LIN {X 0.115,Y -679.979,Z 928.446,A 0.000,B 0.000,C 90.000,E1 296.309} C_DIS
LIN {X -0.394,Y -681.905,Z 928.440,A 0.000,B 0.000,C 90.000,E1 295.155} C_DIS
LIN {X 0.151,Y -683.265,Z 928.434,A 0.000,B 0.000,C 90.000,E1 294.155} C_DIS
LIN {X 0.090,Y -684.389,Z 928.429,A 0.000,B 0.000,C 90.000,E1 293.206} C_DIS
LIN {X -0.388,Y -684.559,Z 928.426,A 0.000,B 0.000,C 90.000,E1 292.770} C_DIS
LIN {X -0.179,Y -684.600,Z 928.425,A 0.000,B 0.000,C 90.000,E1 292.514} C_DIS
LIN {X -0.022,Y -683.786,Z 928.422,A 0.000,B 0.000,C 90.000,E1 292.025} C_DIS
LIN {X 0.182,Y -683.293,Z 928.421,A 0.000,B 0.000,C 90.000,E1 291.770} C_DIS
LIN {X 0.031,Y -682.793,Z 928.420,A 0.000,B 0.000,C 90.000,E1 291.663} C_DIS
LIN {X 0.133,Y -682.008,Z 928.420,A 0.000,B 0.000,C 90.000,E1 291.535} C_DIS
LIN {X -0.294,Y -677.350,Z 928.417,A 0.000,B 0.000,C 90.000,E1 291.099} C_DIS
LIN {X -0.020,Y -676.163,Z 928.417,A 0.000,B 0.000,C 90.000,E1 290.972} C_DIS
LIN {X -0.216,Y -672.859,Z 928.415,A 0.000,B 0.000,C 90.000,E1 290.791} C_DIS
LIN {X 0.088,Y -663.665,Z 928.413,A 0.000,B 0.000,C 90.000,E1 290.248} C_DIS
LIN {X -0.132,Y -662.068,Z 928.412,A 0.000,B 0.000,C 90.000,E1 290.120} C_DIS
LIN {X -0.175,Y -662.057,Z 928.412,A 0.000,B 0.000,C 90.000,E1 290.120} C_DIS
LIN {X -0.103,Y -661.805,Z 928.411,A 0.000,B 0.000,C 90.000,E1 289.939} C_DIS
LIN {X 0.025,Y -662.671,Z 928.408,A 0.000,B 0.000,C 90.000,E1 289.504} C_DIS
LIN {X -0.122,Y -665.204,Z 928.405,A 0.000,B 0.000,C 90.000,E1 288.906} C_DIS
LIN {X -0.022,Y -671.493,Z 928.398,A 0.000,B 0.000,C 90.000,E1 287.692} C_DIS
LIN {X -0.225,Y -674.954,Z 928.394,A 0.000,B 0.000,C 90.000,E1 286.985} C_DIS
LIN {X -0.146,Y -676.936,Z 928.392,A 0.000,B 0.000,C 90.000,E1 286.496} C_DIS
LIN {X -0.291,Y -679.446,Z 928.388,A 0.000,B 0.000,C 90.000,E1 285.788} C_DIS
LIN {X -0.230,Y -681.318,Z 928.384,A 0.000,B 0.000,C 90.000,E1 285.064} C_DIS
LIN {X 0.301,Y -683.455,Z 928.378,A 0.000,B 0.000,C 90.000,E1 284.064} C_DIS
LIN {X 0.201,Y -685.101,Z 928.373,A 0.000,B 0.000,C 90.000,E1 283.119} C_DIS
LIN {X 0.136,Y -686.117,Z 928.369,A 0.000,B 0.000,C 90.000,E1 282.411} C_DIS
LIN {X -0.066,Y -686.891,Z 928.365,A 0.000,B 0.000,C 90.000,E1 281.715} C_DIS
LIN {X -0.102,Y -687.225,Z 928.362,A 0.000,B 0.000,C 90.000,E1 281.243} C_DIS
LIN {X -0.268,Y -687.192,Z 928.360,A 0.000,B 0.000,C 90.000,E1 280.782} C_DIS
LIN {X 0.349,Y -686.686,Z 928.356,A 0.000,B 0.000,C 90.000,E1 280.018} C_DIS
LIN {X 0.186,Y -685.782,Z 928.353,A 0.000,B 0.000,C 90.000,E1 279.557} C_DIS
LIN {X 0.022,Y -684.420,Z 928.351,A 0.000,B 0.000,C 90.000,E1 279.095} C_DIS
LIN {X -0.009,Y -683.605,Z 928.349,A 0.000,B 0.000,C 90.000,E1 278.859} C_DIS
LIN {X -0.183,Y -681.661,Z 928.347,A 0.000,B 0.000,C 90.000,E1 278.398} C_DIS
LIN {X 0.124,Y -676.310,Z 928.341,A 0.000,B 0.000,C 90.000,E1 277.296} C_DIS
LIN {X -0.253,Y -671.792,Z 928.336,A 0.000,B 0.000,C 90.000,E1 276.486} C_DIS
LIN {X 0.079,Y -668.243,Z 928.333,A 0.000,B 0.000,C 90.000,E1 275.853} C_DIS
LIN {X -0.280,Y -664.000,Z 928.329,A 0.000,B 0.000,C 90.000,E1 275.277} C_DIS
LIN {X 0.079,Y -660.284,Z 928.327,A 0.000,B 0.000,C 90.000,E1 274.759} C_DIS
LIN {X 0.260,Y -655.075,Z 928.323,A 0.000,B 0.000,C 90.000,E1 274.131} C_DIS
LIN {X -0.097,Y -650.616,Z 928.320,A 0.000,B 0.000,C 90.000,E1 273.669} C_DIS
LIN {X 0.179,Y -644.503,Z 928.317,A 0.000,B 0.000,C 90.000,E1 273.037} C_DIS
LIN {X 0.014,Y -637.880,Z 928.314,A 0.000,B 0.000,C 90.000,E1 272.465} C_DIS
LIN {X 0.210,Y -630.842,Z 928.311,A 0.000,B 0.000,C 90.000,E1 271.892} C_DIS
LIN {X 0.177,Y -623.249,Z 928.308,A 0.000,B 0.000,C 90.000,E1 271.375} C_DIS
LIN {X -0.081,Y -615.438,Z 928.305,A 0.000,B 0.000,C 90.000,E1 270.917} C_DIS
LIN {X 0.026,Y -610.795,Z 928.304,A 0.000,B 0.000,C 90.000,E1 270.630} C_DIS
LIN {X 0.019,Y -604.204,Z 928.302,A 0.000,B 0.000,C 90.000,E1 270.286} C_DIS
LIN {X 0.254,Y -597.487,Z 928.300,A 0.000,B 0.000,C 90.000,E1 269.943} C_DIS
LIN {X 0.204,Y -590.404,Z 928.298,A 0.000,B 0.000,C 90.000,E1 269.656} C_DIS
LIN {X -0.043,Y -585.027,Z 928.297,A 0.000,B 0.000,C 90.000,E1 269.484} C_DIS
LIN {X -0.044,Y -577.197,Z 928.296,A 0.000,B 0.000,C 90.000,E1 269.255} C_DIS
LIN {X 0.274,Y -571.267,Z 928.295,A 0.000,B 0.000,C 90.000,E1 269.083} C_DIS
LIN {X -0.226,Y -565.261,Z 928.294,A 0.000,B 0.000,C 90.000,E1 269.026} C_DIS
LIN {X 0.072,Y -557.427,Z 928.294,A 0.000,B 0.000,C 90.000,E1 268.912} C_DIS
LIN {X 0.257,Y -552.326,Z 928.294,A 0.000,B 0.000,C 90.000,E1 268.854} C_DIS
LIN {X -0.168,Y -550.890,Z 928.294,A 0.000,B 0.000,C 90.000,E1 268.854} C_DIS
LIN {X -0.201,Y -550.829,Z 928.294,A 0.000,B 0.000,C 90.000,E1 268.854} C_DIS
LIN {X 0.151,Y -550.326,Z 928.293,A 0.000,B 0.000,C 90.000,E1 268.740} C_DIS
LIN {X 0.155,Y -546.076,Z 928.290,A 0.000,B 0.000,C 90.000,E1 268.224} C_DIS
LIN {X 0.133,Y -544.236,Z 928.289,A 0.000,B 0.000,C 90.000,E1 268.051} C_DIS
LIN {X 0.091,Y -544.197,Z 928.289,A 0.000,B 0.000,C 90.000,E1 268.051} C_DIS
LIN {X -0.037,Y -543.551,Z 928.288,A 0.000,B 0.000,C 90.000,E1 267.822} C_DIS
LIN {X 0.095,Y -542.151,Z 928.281,A 0.000,B 0.000,C 90.000,E1 266.617} C_DIS
LIN {X -0.169,Y -540.126,Z 928.267,A 0.000,B 0.000,C 90.000,E1 264.090} C_DIS
LIN {X 0.086,Y -538.982,Z 928.258,A 0.000,B 0.000,C 90.000,E1 262.356} C_DIS
LIN {X -0.281,Y -537.936,Z 928.250,A 0.000,B 0.000,C 90.000,E1 260.971} C_DIS
LIN {X -0.091,Y -537.174,Z 928.245,A 0.000,B 0.000,C 90.000,E1 260.095} C_DIS
LIN {X 0.097,Y -536.165,Z 928.240,A 0.000,B 0.000,C 90.000,E1 259.218} C_DIS
LIN {X 0.064,Y -532.655,Z 928.226,A 0.000,B 0.000,C 90.000,E1 256.645} C_DIS
LIN {X 0.087,Y -530.180,Z 928.215,A 0.000,B 0.000,C 90.000,E1 254.629} C_DIS
LIN {X 0.023,Y -528.110,Z 928.205,A 0.000,B 0.000,C 90.000,E1 252.906} C_DIS
LIN {X 0.055,Y -526.299,Z 928.197,A 0.000,B 0.000,C 90.000,E1 251.456} C_DIS
LIN {X 0.053,Y -523.295,Z 928.184,A 0.000,B 0.000,C 90.000,E1 249.135} C_DIS
LIN {X -0.153,Y -520.997,Z 928.174,A 0.000,B 0.000,C 90.000,E1 247.411} C_DIS
LIN {X 0.115,Y -518.888,Z 928.166,A 0.000,B 0.000,C 90.000,E1 245.921} C_DIS
LIN {X 0.212,Y -516.133,Z 928.157,A 0.000,B 0.000,C 90.000,E1 244.152} C_DIS
LIN {X 0.121,Y -513.836,Z 928.148,A 0.000,B 0.000,C 90.000,E1 242.692} C_DIS
LIN {X -0.235,Y -511.323,Z 928.140,A 0.000,B 0.000,C 90.000,E1 241.257} C_DIS
LIN {X -0.017,Y -509.278,Z 928.134,A 0.000,B 0.000,C 90.000,E1 240.049} C_DIS
LIN {X 0.242,Y -506.592,Z 928.125,A 0.000,B 0.000,C 90.000,E1 238.535} C_DIS
LIN {X -0.036,Y -504.197,Z 928.119,A 0.000,B 0.000,C 90.000,E1 237.375} C_DIS
LIN {X 0.071,Y -501.549,Z 928.112,A 0.000,B 0.000,C 90.000,E1 236.167} C_DIS
LIN {X -0.116,Y -496.120,Z 928.099,A 0.000,B 0.000,C 90.000,E1 233.783} C_DIS
LIN {X -0.109,Y -491.517,Z 928.087,A 0.000,B 0.000,C 90.000,E1 231.662} C_DIS
LIN {X 0.122,Y -489.459,Z 928.082,A 0.000,B 0.000,C 90.000,E1 230.723} C_DIS
LIN {X -0.248,Y -485.323,Z 928.072,A 0.000,B 0.000,C 90.000,E1 228.933} C_DIS
LIN {X -0.204,Y -481.829,Z 928.063,A 0.000,B 0.000,C 90.000,E1 227.391} C_DIS
LIN {X 0.219,Y -477.697,Z 928.053,A 0.000,B 0.000,C 90.000,E1 225.486} C_DIS
LIN {X -0.003,Y -475.046,Z 928.046,A 0.000,B 0.000,C 90.000,E1 224.271} C_DIS
LIN {X -0.061,Y -470.852,Z 928.036,A 0.000,B 0.000,C 90.000,E1 222.405} C_DIS
LIN {X -0.047,Y -468.121,Z 928.029,A 0.000,B 0.000,C 90.000,E1 221.148} C_DIS
LIN {X -0.019,Y -461.957,Z 928.013,A 0.000,B 0.000,C 90.000,E1 218.302} C_DIS
LIN {X -0.020,Y -459.252,Z 928.006,A 0.000,B 0.000,C 90.000,E1 217.030} C_DIS
LIN {X -0.056,Y -455.812,Z 927.997,A 0.000,B 0.000,C 90.000,E1 215.438} C_DIS
LIN {X 0.030,Y -451.538,Z 927.986,A 0.000,B 0.000,C 90.000,E1 213.499} C_DIS
LIN {X 0.151,Y -447.320,Z 927.975,A 0.000,B 0.000,C 90.000,E1 211.544} C_DIS
LIN {X 0.105,Y -440.899,Z 927.959,A 0.000,B 0.000,C 90.000,E1 208.615} C_DIS
LIN {X -0.144,Y -438.025,Z 927.952,A 0.000,B 0.000,C 90.000,E1 207.334} C_DIS
LIN {X -0.020,Y -434.378,Z 927.943,A 0.000,B 0.000,C 90.000,E1 205.668} C_DIS
LIN {X 0.038,Y -429.286,Z 927.930,A 0.000,B 0.000,C 90.000,E1 203.334} C_DIS
LIN {X -0.174,Y -426.387,Z 927.922,A 0.000,B 0.000,C 90.000,E1 202.025} C_DIS
LIN {X 0.144,Y -422.679,Z 927.913,A 0.000,B 0.000,C 90.000,E1 200.301} C_DIS
LIN {X -0.033,Y -416.572,Z 927.896,A 0.000,B 0.000,C 90.000,E1 197.275} C_DIS
LIN {X -0.090,Y -414.522,Z 927.890,A 0.000,B 0.000,C 90.000,E1 196.260} C_DIS
LIN {X -0.012,Y -410.975,Z 927.881,A 0.000,B 0.000,C 90.000,E1 194.537} C_DIS
LIN {X -0.124,Y -408.214,Z 927.873,A 0.000,B 0.000,C 90.000,E1 193.175} C_DIS
LIN {X 0.121,Y -403.378,Z 927.860,A 0.000,B 0.000,C 90.000,E1 190.715} C_DIS
LIN {X 0.076,Y -398.649,Z 927.846,A 0.000,B 0.000,C 90.000,E1 188.276} C_DIS
LIN {X 0.182,Y -393.790,Z 927.832,A 0.000,B 0.000,C 90.000,E1 185.796} C_DIS
LIN {X 0.017,Y -388.588,Z 927.817,A 0.000,B 0.000,C 90.000,E1 182.980} C_DIS
LIN {X 0.071,Y -382.269,Z 927.795,A 0.000,B 0.000,C 90.000,E1 179.026} C_DIS
LIN {X 0.116,Y -381.021,Z 927.789,A 0.000,B 0.000,C 90.000,E1 177.936} C_DIS
LIN {X 0.130,Y -380.155,Z 927.783,A 0.000,B 0.000,C 90.000,E1 176.849} C_DIS
LIN {X -0.103,Y -380.088,Z 927.779,A 0.000,B 0.000,C 90.000,E1 176.159} C_DIS
LIN {X 0.044,Y -380.506,Z 927.775,A 0.000,B 0.000,C 90.000,E1 175.412} C_DIS
LIN {X -0.055,Y -381.032,Z 927.773,A 0.000,B 0.000,C 90.000,E1 175.065} C_DIS
LIN {X -0.179,Y -382.141,Z 927.770,A 0.000,B 0.000,C 90.000,E1 174.609} C_DIS
LIN {X -0.206,Y -384.369,Z 927.767,A 0.000,B 0.000,C 90.000,E1 174.033} C_DIS
LIN {X -0.085,Y -386.614,Z 927.765,A 0.000,B 0.000,C 90.000,E1 173.628} C_DIS
LIN {X -0.161,Y -389.018,Z 927.763,A 0.000,B 0.000,C 90.000,E1 173.280} C_DIS
LIN {X -0.073,Y -391.403,Z 927.761,A 0.000,B 0.000,C 90.000,E1 172.989} C_DIS
LIN {X 0.127,Y -395.578,Z 927.759,A 0.000,B 0.000,C 90.000,E1 172.534} C_DIS
LIN {X 0.119,Y -403.599,Z 927.755,A 0.000,B 0.000,C 90.000,E1 171.894} C_DIS
LIN {X 0.216,Y -413.105,Z 927.751,A 0.000,B 0.000,C 90.000,E1 171.197} C_DIS
LIN {X -0.058,Y -424.372,Z 927.747,A 0.000,B 0.000,C 90.000,E1 170.387} C_DIS
LIN {X 0.074,Y -433.736,Z 927.742,A 0.000,B 0.000,C 90.000,E1 169.634} C_DIS
LIN {X -0.122,Y -438.390,Z 927.740,A 0.000,B 0.000,C 90.000,E1 169.285} C_DIS
LIN {X -0.153,Y -445.924,Z 927.737,A 0.000,B 0.000,C 90.000,E1 168.634} C_DIS
LIN {X 0.139,Y -453.234,Z 927.733,A 0.000,B 0.000,C 90.000,E1 167.937} C_DIS
LIN {X -0.032,Y -461.903,Z 927.728,A 0.000,B 0.000,C 90.000,E1 167.117} C_DIS
LIN {X -0.138,Y -468.940,Z 927.724,A 0.000,B 0.000,C 90.000,E1 166.408} C_DIS
LIN {X -0.197,Y -476.850,Z 927.719,A 0.000,B 0.000,C 90.000,E1 165.519} C_DIS
LIN {X -0.177,Y -486.002,Z 927.714,A 0.000,B 0.000,C 90.000,E1 164.448} C_DIS
LIN {X -0.166,Y -491.991,Z 927.709,A 0.000,B 0.000,C 90.000,E1 163.685} C_DIS
LIN {X 0.049,Y -499.996,Z 927.703,A 0.000,B 0.000,C 90.000,E1 162.598} C_DIS
LIN {X 0.223,Y -512.447,Z 927.693,A 0.000,B 0.000,C 90.000,E1 160.786} C_DIS
LIN {X 0.067,Y -520.436,Z 927.687,A 0.000,B 0.000,C 90.000,E1 159.625} C_DIS
LIN {X 0.022,Y -527.959,Z 927.680,A 0.000,B 0.000,C 90.000,E1 158.465} C_DIS
LIN {X 0.077,Y -535.176,Z 927.674,A 0.000,B 0.000,C 90.000,E1 157.305} C_DIS
LIN {X 0.045,Y -544.769,Z 927.665,A 0.000,B 0.000,C 90.000,E1 155.741} C_DIS
LIN {X -0.333,Y -550.536,Z 927.660,A 0.000,B 0.000,C 90.000,E1 154.793} C_DIS
LIN {X -0.120,Y -557.640,Z 927.653,A 0.000,B 0.000,C 90.000,E1 153.512} C_DIS
LIN {X 0.211,Y -564.128,Z 927.646,A 0.000,B 0.000,C 90.000,E1 152.231} C_DIS
LIN {X -0.076,Y -566.272,Z 927.644,A 0.000,B 0.000,C 90.000,E1 151.847} C_DIS
LIN {X -0.092,Y -574.176,Z 927.634,A 0.000,B 0.000,C 90.000,E1 150.205} C_DIS
LIN {X -0.226,Y -579.539,Z 927.628,A 0.000,B 0.000,C 90.000,E1 148.997} C_DIS
LIN {X -0.226,Y -581.876,Z 927.625,A 0.000,B 0.000,C 90.000,E1 148.456} C_DIS
LIN {X -0.128,Y -588.414,Z 927.616,A 0.000,B 0.000,C 90.000,E1 146.834} C_DIS
LIN {X 0.007,Y -592.718,Z 927.610,A 0.000,B 0.000,C 90.000,E1 145.754} C_DIS
LIN {X 0.045,Y -596.901,Z 927.604,A 0.000,B 0.000,C 90.000,E1 144.689} C_DIS
LIN {X -0.094,Y -599.878,Z 927.599,A 0.000,B 0.000,C 90.000,E1 143.909} C_DIS
LIN {X 0.084,Y -605.610,Z 927.591,A 0.000,B 0.000,C 90.000,E1 142.316} C_DIS
LIN {X -0.193,Y -612.532,Z 927.581,A 0.000,B 0.000,C 90.000,E1 140.517} C_DIS
LIN {X 0.155,Y -618.534,Z 927.572,A 0.000,B 0.000,C 90.000,E1 138.933} C_DIS
LIN {X 0.089,Y -628.640,Z 927.558,A 0.000,B 0.000,C 90.000,E1 136.377} C_DIS
LIN {X 0.058,Y -632.754,Z 927.552,A 0.000,B 0.000,C 90.000,E1 135.364} C_DIS
LIN {X -0.115,Y -638.687,Z 927.544,A 0.000,B 0.000,C 90.000,E1 133.866} C_DIS
LIN {X -0.004,Y -642.636,Z 927.538,A 0.000,B 0.000,C 90.000,E1 132.852} C_DIS
LIN {X -0.049,Y -650.428,Z 927.527,A 0.000,B 0.000,C 90.000,E1 130.862} C_DIS
LIN {X -0.261,Y -655.186,Z 927.520,A 0.000,B 0.000,C 90.000,E1 129.644} C_DIS
LIN {X 0.130,Y -661.759,Z 927.511,A 0.000,B 0.000,C 90.000,E1 127.890} C_DIS
LIN {X 0.166,Y -667.284,Z 927.503,A 0.000,B 0.000,C 90.000,E1 126.423} C_DIS
LIN {X -0.080,Y -671.674,Z 927.496,A 0.000,B 0.000,C 90.000,E1 125.231} C_DIS
LIN {X 0.148,Y -674.922,Z 927.490,A 0.000,B 0.000,C 90.000,E1 124.246} C_DIS
LIN {X 0.438,Y -677.247,Z 927.486,A 0.000,B 0.000,C 90.000,E1 123.499} C_DIS
LIN {X -0.183,Y -679.386,Z 927.482,A 0.000,B 0.000,C 90.000,E1 122.832} C_DIS
LIN {X 0.323,Y -682.523,Z 927.476,A 0.000,B 0.000,C 90.000,E1 121.592} C_DIS
LIN {X -0.043,Y -684.633,Z 927.470,A 0.000,B 0.000,C 90.000,E1 120.669} C_DIS
LIN {X -0.001,Y -686.108,Z 927.466,A 0.000,B 0.000,C 90.000,E1 119.951} C_DIS
LIN {X 0.019,Y -687.763,Z 927.461,A 0.000,B 0.000,C 90.000,E1 118.999} C_DIS
LIN {X 0.089,Y -688.867,Z 927.457,A 0.000,B 0.000,C 90.000,E1 118.281} C_DIS
LIN {X 0.084,Y -689.911,Z 927.452,A 0.000,B 0.000,C 90.000,E1 117.334} C_DIS
LIN {X -0.203,Y -690.487,Z 927.447,A 0.000,B 0.000,C 90.000,E1 116.411} C_DIS
LIN {X 0.206,Y -690.666,Z 927.443,A 0.000,B 0.000,C 90.000,E1 115.668} C_DIS
LIN {X 0.241,Y -690.715,Z 927.438,A 0.000,B 0.000,C 90.000,E1 114.719} C_DIS
LIN {X 0.038,Y -690.480,Z 927.434,A 0.000,B 0.000,C 90.000,E1 114.027} C_DIS
LIN {X -0.125,Y -690.060,Z 927.431,A 0.000,B 0.000,C 90.000,E1 113.567} C_DIS
LIN {X -0.168,Y -689.627,Z 927.430,A 0.000,B 0.000,C 90.000,E1 113.334} C_DIS
LIN {X 0.290,Y -688.240,Z 927.427,A 0.000,B 0.000,C 90.000,E1 112.823} C_DIS
LIN {X 0.137,Y -687.716,Z 927.426,A 0.000,B 0.000,C 90.000,E1 112.717} C_DIS
LIN {X -0.059,Y -684.321,Z 927.424,A 0.000,B 0.000,C 90.000,E1 112.259} C_DIS
LIN {X -0.211,Y -683.240,Z 927.423,A 0.000,B 0.000,C 90.000,E1 112.153} C_DIS
LIN {X -0.108,Y -681.860,Z 927.422,A 0.000,B 0.000,C 90.000,E1 112.025} C_DIS
LIN {X -0.005,Y -679.584,Z 927.422,A 0.000,B 0.000,C 90.000,E1 111.897} C_DIS
LIN {X 0.194,Y -674.984,Z 927.421,A 0.000,B 0.000,C 90.000,E1 111.716} C_DIS
LIN {X 0.300,Y -669.777,Z 927.420,A 0.000,B 0.000,C 90.000,E1 111.535} C_DIS
LIN {X -0.371,Y -666.947,Z 927.419,A 0.000,B 0.000,C 90.000,E1 111.535} C_DIS
LIN {X -0.229,Y -659.882,Z 927.419,A 0.000,B 0.000,C 90.000,E1 111.461} C_DIS
LIN {X 0.340,Y -652.708,Z 927.419,A 0.000,B 0.000,C 90.000,E1 111.408} C_DIS
LIN {X 0.295,Y -643.253,Z 927.419,A 0.000,B 0.000,C 90.000,E1 111.408} C_DIS
LIN {X -0.011,Y -638.058,Z 927.419,A 0.000,B 0.000,C 90.000,E1 111.408} C_DIS
LIN {X 0.198,Y -634.455,Z 927.419,A 0.000,B 0.000,C 90.000,E1 111.354} C_DIS
LIN {X 0.110,Y -629.194,Z 927.418,A 0.000,B 0.000,C 90.000,E1 111.280} C_DIS
LIN {X -0.190,Y -621.802,Z 927.417,A 0.000,B 0.000,C 90.000,E1 111.153} C_DIS
LIN {X 0.094,Y -614.447,Z 927.416,A 0.000,B 0.000,C 90.000,E1 110.918} C_DIS
LIN {X -0.134,Y -606.224,Z 927.414,A 0.000,B 0.000,C 90.000,E1 110.610} C_DIS
LIN {X -0.176,Y -603.378,Z 927.414,A 0.000,B 0.000,C 90.000,E1 110.482} C_DIS
LIN {X 0.115,Y -598.239,Z 927.412,A 0.000,B 0.000,C 90.000,E1 110.174} C_DIS
LIN {X -0.185,Y -590.045,Z 927.409,A 0.000,B 0.000,C 90.000,E1 109.685} C_DIS
LIN {X -0.322,Y -583.118,Z 927.407,A 0.000,B 0.000,C 90.000,E1 109.214} C_DIS
LIN {X -0.218,Y -578.724,Z 927.405,A 0.000,B 0.000,C 90.000,E1 108.906} C_DIS
LIN {X 0.107,Y -571.680,Z 927.403,A 0.000,B 0.000,C 90.000,E1 108.489} C_DIS
LIN {X 0.028,Y -564.876,Z 927.401,A 0.000,B 0.000,C 90.000,E1 108.181} C_DIS
LIN {X 0.222,Y -557.773,Z 927.399,A 0.000,B 0.000,C 90.000,E1 107.873} C_DIS
LIN {X -0.079,Y -554.844,Z 927.399,A 0.000,B 0.000,C 90.000,E1 107.764} C_DIS
LIN {X 0.048,Y -552.961,Z 927.398,A 0.000,B 0.000,C 90.000,E1 107.583} C_DIS
LIN {X 0.010,Y -552.942,Z 927.398,A 0.000,B 0.000,C 90.000,E1 107.583} C_DIS
LIN {X 0.136,Y -552.516,Z 927.396,A 0.000,B 0.000,C 90.000,E1 107.330} C_DIS
LIN {X 0.117,Y -552.658,Z 927.392,A 0.000,B 0.000,C 90.000,E1 106.622} C_DIS
LIN {X -0.196,Y -553.186,Z 927.386,A 0.000,B 0.000,C 90.000,E1 105.536} C_DIS
LIN {X 0.116,Y -553.904,Z 927.377,A 0.000,B 0.000,C 90.000,E1 103.828} C_DIS
LIN {X 0.034,Y -555.068,Z 927.366,A 0.000,B 0.000,C 90.000,E1 101.883} C_DIS
LIN {X -0.115,Y -556.765,Z 927.354,A 0.000,B 0.000,C 90.000,E1 99.670} C_DIS
LIN {X -0.083,Y -557.816,Z 927.346,A 0.000,B 0.000,C 90.000,E1 98.276} C_DIS
LIN {X -0.112,Y -558.880,Z 927.338,A 0.000,B 0.000,C 90.000,E1 96.891} C_DIS
LIN {X -0.048,Y -559.931,Z 927.329,A 0.000,B 0.000,C 90.000,E1 95.220} C_DIS
LIN {X -0.098,Y -560.701,Z 927.321,A 0.000,B 0.000,C 90.000,E1 93.841} C_DIS
LIN {X -0.168,Y -561.417,Z 927.314,A 0.000,B 0.000,C 90.000,E1 92.465} C_DIS
LIN {X -0.127,Y -562.099,Z 927.304,A 0.000,B 0.000,C 90.000,E1 90.802} C_DIS
LIN {X 0.278,Y -562.437,Z 927.298,A 0.000,B 0.000,C 90.000,E1 89.656} C_DIS
LIN {X 0.222,Y -562.782,Z 927.291,A 0.000,B 0.000,C 90.000,E1 88.282} C_DIS
LIN {X 0.184,Y -563.045,Z 927.283,A 0.000,B 0.000,C 90.000,E1 86.906} C_DIS
LIN {X 0.088,Y -563.269,Z 927.277,A 0.000,B 0.000,C 90.000,E1 85.812} C_DIS
LIN {X 0.195,Y -563.518,Z 927.268,A 0.000,B 0.000,C 90.000,E1 84.147} C_DIS
LIN {X -0.053,Y -563.868,Z 927.257,A 0.000,B 0.000,C 90.000,E1 82.243} C_DIS
LIN {X -0.215,Y -564.420,Z 927.246,A 0.000,B 0.000,C 90.000,E1 80.330} C_DIS
LIN {X -0.273,Y -565.235,Z 927.235,A 0.000,B 0.000,C 90.000,E1 78.409} C_DIS
LIN {X 0.309,Y -566.172,Z 927.226,A 0.000,B 0.000,C 90.000,E1 76.700} C_DIS
LIN {X -0.178,Y -567.199,Z 927.217,A 0.000,B 0.000,C 90.000,E1 75.102} C_DIS
LIN {X -0.273,Y -567.944,Z 927.210,A 0.000,B 0.000,C 90.000,E1 73.740} C_DIS
LIN {X -0.201,Y -568.651,Z 927.202,A 0.000,B 0.000,C 90.000,E1 72.362} C_DIS
LIN {X 0.217,Y -569.361,Z 927.193,A 0.000,B 0.000,C 90.000,E1 70.678} C_DIS
LIN {X -0.200,Y -569.731,Z 927.187,A 0.000,B 0.000,C 90.000,E1 69.625} C_DIS
LIN {X 0.073,Y -570.204,Z 927.179,A 0.000,B 0.000,C 90.000,E1 68.230} C_DIS
LIN {X -0.152,Y -570.492,Z 927.170,A 0.000,B 0.000,C 90.000,E1 66.613} C_DIS
LIN {X -0.137,Y -570.712,Z 927.161,A 0.000,B 0.000,C 90.000,E1 64.973} C_DIS
LIN {X -0.121,Y -570.936,Z 927.152,A 0.000,B 0.000,C 90.000,E1 63.332} C_DIS
LIN {X -0.095,Y -570.934,Z 927.143,A 0.000,B 0.000,C 90.000,E1 61.691} C_DIS
LIN {X -0.051,Y -570.926,Z 927.134,A 0.000,B 0.000,C 90.000,E1 60.049} C_DIS
LIN {X -0.020,Y -570.829,Z 927.125,A 0.000,B 0.000,C 90.000,E1 58.408} C_DIS
LIN {X -0.012,Y -570.380,Z 927.117,A 0.000,B 0.000,C 90.000,E1 57.041} C_DIS
LIN {X -0.136,Y -569.914,Z 927.111,A 0.000,B 0.000,C 90.000,E1 55.960} C_DIS
LIN {X 0.245,Y -569.455,Z 927.106,A 0.000,B 0.000,C 90.000,E1 55.102} C_DIS
LIN {X -0.164,Y -568.917,Z 927.102,A 0.000,B 0.000,C 90.000,E1 54.322} C_DIS
LIN {X -0.120,Y -568.294,Z 927.097,A 0.000,B 0.000,C 90.000,E1 53.497} C_DIS
LIN {X 0.250,Y -567.516,Z 927.093,A 0.000,B 0.000,C 90.000,E1 52.637} C_DIS
LIN {X 0.280,Y -566.284,Z 927.087,A 0.000,B 0.000,C 90.000,E1 51.537} C_DIS
LIN {X 0.184,Y -565.204,Z 927.082,A 0.000,B 0.000,C 90.000,E1 50.723} C_DIS
LIN {X 0.181,Y -563.563,Z 927.076,A 0.000,B 0.000,C 90.000,E1 49.622} C_DIS
LIN {X 0.092,Y -561.541,Z 927.070,A 0.000,B 0.000,C 90.000,E1 48.528} C_DIS
LIN {X -0.060,Y -559.808,Z 927.065,A 0.000,B 0.000,C 90.000,E1 47.715} C_DIS
LIN {X 0.065,Y -558.557,Z 927.062,A 0.000,B 0.000,C 90.000,E1 47.148} C_DIS
LIN {X -0.089,Y -555.568,Z 927.056,A 0.000,B 0.000,C 90.000,E1 46.053} C_DIS
LIN {X 0.011,Y -553.938,Z 927.053,A 0.000,B 0.000,C 90.000,E1 45.486} C_DIS
LIN {X -0.250,Y -551.170,Z 927.048,A 0.000,B 0.000,C 90.000,E1 44.676} C_DIS
LIN {X -0.180,Y -549.162,Z 927.045,A 0.000,B 0.000,C 90.000,E1 44.109} C_DIS
LIN {X -0.095,Y -545.833,Z 927.040,A 0.000,B 0.000,C 90.000,E1 43.257} C_DIS
LIN {X -0.264,Y -544.054,Z 927.038,A 0.000,B 0.000,C 90.000,E1 42.852} C_DIS
LIN {X -0.063,Y -540.785,Z 927.034,A 0.000,B 0.000,C 90.000,E1 42.123} C_DIS
LIN {X -0.038,Y -537.972,Z 927.031,A 0.000,B 0.000,C 90.000,E1 41.553} C_DIS
LIN {X 0.095,Y -534.170,Z 927.027,A 0.000,B 0.000,C 90.000,E1 40.825} C_DIS
LIN {X -0.086,Y -531.769,Z 927.025,A 0.000,B 0.000,C 90.000,E1 40.415} C_DIS
LIN {X -0.048,Y -525.603,Z 927.019,A 0.000,B 0.000,C 90.000,E1 39.402} C_DIS
LIN {X -0.160,Y -520.015,Z 927.014,A 0.000,B 0.000,C 90.000,E1 38.543} C_DIS
LIN {X 0.054,Y -516.102,Z 927.011,A 0.000,B 0.000,C 90.000,E1 37.935} C_DIS
LIN {X -0.158,Y -509.901,Z 927.006,A 0.000,B 0.000,C 90.000,E1 37.076} C_DIS
LIN {X 0.217,Y -504.234,Z 927.002,A 0.000,B 0.000,C 90.000,E1 36.297} C_DIS
LIN {X -0.091,Y -500.675,Z 926.999,A 0.000,B 0.000,C 90.000,E1 35.884} C_DIS
LIN {X 0.087,Y -495.610,Z 926.996,A 0.000,B 0.000,C 90.000,E1 35.264} C_DIS
LIN {X -0.153,Y -487.475,Z 926.991,A 0.000,B 0.000,C 90.000,E1 34.405} C_DIS
LIN {X -0.150,Y -481.790,Z 926.988,A 0.000,B 0.000,C 90.000,E1 33.833} C_DIS
LIN {X 0.297,Y -474.576,Z 926.984,A 0.000,B 0.000,C 90.000,E1 33.086} C_DIS
LIN {X 0.150,Y -465.595,Z 926.980,A 0.000,B 0.000,C 90.000,E1 32.291} C_DIS
LIN {X -0.185,Y -458.095,Z 926.976,A 0.000,B 0.000,C 90.000,E1 31.671} C_DIS
LIN {X 0.185,Y -445.882,Z 926.970,A 0.000,B 0.000,C 90.000,E1 30.590} C_DIS
LIN {X -0.078,Y -427.545,Z 926.962,A 0.000,B 0.000,C 90.000,E1 29.077} C_DIS
LIN {X -0.079,Y -411.032,Z 926.953,A 0.000,B 0.000,C 90.000,E1 27.590} C_DIS
LIN {X -0.105,Y -399.220,Z 926.947,A 0.000,B 0.000,C 90.000,E1 26.411} C_DIS
LIN {X 0.139,Y -393.877,Z 926.943,A 0.000,B 0.000,C 90.000,E1 25.720} C_DIS
LIN {X -0.092,Y -391.681,Z 926.941,A 0.000,B 0.000,C 90.000,E1 25.387} C_DIS
LIN {X 0.073,Y -390.903,Z 926.940,A 0.000,B 0.000,C 90.000,E1 25.207} C_DIS
LIN {X 0.059,Y -389.640,Z 926.938,A 0.000,B 0.000,C 90.000,E1 24.823} C_DIS
LIN {X -0.098,Y -388.977,Z 926.935,A 0.000,B 0.000,C 90.000,E1 24.335} C_DIS
LIN {X -0.161,Y -388.740,Z 926.931,A 0.000,B 0.000,C 90.000,E1 23.643} C_DIS
LIN {X 0.048,Y -388.993,Z 926.927,A 0.000,B 0.000,C 90.000,E1 22.898} C_DIS
LIN {X 0.226,Y -392.983,Z 926.904,A 0.000,B 0.000,C 90.000,E1 18.598} C_DIS
LIN {X 0.127,Y -395.874,Z 926.890,A 0.000,B 0.000,C 90.000,E1 16.134} C_DIS
LIN {X -0.182,Y -398.593,Z 926.878,A 0.000,B 0.000,C 90.000,E1 14.064} C_DIS
LIN {X -0.062,Y -402.673,Z 926.862,A 0.000,B 0.000,C 90.000,E1 11.243} C_DIS
LIN {X -0.049,Y -406.553,Z 926.849,A 0.000,B 0.000,C 90.000,E1 8.803} C_DIS
LIN {X 0.023,Y -412.139,Z 926.832,A 0.000,B 0.000,C 90.000,E1 5.682} C_DIS
LIN {X 0.179,Y -418.345,Z 926.815,A 0.000,B 0.000,C 90.000,E1 2.579} C_DIS
LIN {X 0.161,Y -424.773,Z 926.799,A 0.000,B 0.000,C 90.000,E1 359.771} C_DIS
LIN {X 0.028,Y -428.998,Z 926.790,A 0.000,B 0.000,C 90.000,E1 358.108} C_DIS
LIN {X 0.129,Y -430.673,Z 926.787,A 0.000,B 0.000,C 90.000,E1 357.593} C_DIS
LIN {X -0.090,Y -433.342,Z 926.784,A 0.000,B 0.000,C 90.000,E1 357.078} C_DIS
LIN {X -0.120,Y -435.868,Z 926.782,A 0.000,B 0.000,C 90.000,E1 356.731} C_DIS
LIN {X -0.076,Y -437.355,Z 926.781,A 0.000,B 0.000,C 90.000,E1 356.560} C_DIS
LIN {X 0.054,Y -440.722,Z 926.779,A 0.000,B 0.000,C 90.000,E1 356.274} C_DIS
LIN {X -0.124,Y -446.240,Z 926.778,A 0.000,B 0.000,C 90.000,E1 355.988} C_DIS
LIN {X 0.115,Y -461.474,Z 926.774,A 0.000,B 0.000,C 90.000,E1 355.241} C_DIS
LIN {X -0.222,Y -471.486,Z 926.771,A 0.000,B 0.000,C 90.000,E1 354.780} C_DIS
LIN {X -0.240,Y -485.083,Z 926.767,A 0.000,B 0.000,C 90.000,E1 354.090} C_DIS
LIN {X -0.074,Y -496.657,Z 926.764,A 0.000,B 0.000,C 90.000,E1 353.451} C_DIS
LIN {X -0.209,Y -507.904,Z 926.760,A 0.000,B 0.000,C 90.000,E1 352.818} C_DIS
LIN {X 0.274,Y -519.224,Z 926.756,A 0.000,B 0.000,C 90.000,E1 352.064} C_DIS
LIN {X 0.210,Y -525.403,Z 926.754,A 0.000,B 0.000,C 90.000,E1 351.659} C_DIS
LIN {X 0.124,Y -534.116,Z 926.750,A 0.000,B 0.000,C 90.000,E1 351.027} C_DIS
LIN {X 0.133,Y -541.242,Z 926.747,A 0.000,B 0.000,C 90.000,E1 350.443} C_DIS
LIN {X -0.053,Y -548.013,Z 926.744,A 0.000,B 0.000,C 90.000,E1 349.859} C_DIS
LIN {X 0.134,Y -553.199,Z 926.741,A 0.000,B 0.000,C 90.000,E1 349.342} C_DIS
LIN {X 0.169,Y -558.157,Z 926.738,A 0.000,B 0.000,C 90.000,E1 348.814} C_DIS
LIN {X -0.155,Y -566.334,Z 926.733,A 0.000,B 0.000,C 90.000,E1 347.881} C_DIS
LIN {X 0.065,Y -571.738,Z 926.729,A 0.000,B 0.000,C 90.000,E1 347.173} C_DIS
LIN {X -0.258,Y -579.612,Z 926.723,A 0.000,B 0.000,C 90.000,E1 346.117} C_DIS
LIN {X 0.084,Y -583.994,Z 926.719,A 0.000,B 0.000,C 90.000,E1 345.408} C_DIS
LIN {X 0.149,Y -589.855,Z 926.714,A 0.000,B 0.000,C 90.000,E1 344.464} C_DIS
LIN {X 0.142,Y -596.559,Z 926.707,A 0.000,B 0.000,C 90.000,E1 343.268} C_DIS
LIN {X 0.095,Y -604.628,Z 926.698,A 0.000,B 0.000,C 90.000,E1 341.692} C_DIS
LIN {X 0.253,Y -611.456,Z 926.690,A 0.000,B 0.000,C 90.000,E1 340.242} C_DIS
LIN {X 0.231,Y -615.563,Z 926.685,A 0.000,B 0.000,C 90.000,E1 339.337} C_DIS
LIN {X -0.365,Y -621.054,Z 926.678,A 0.000,B 0.000,C 90.000,E1 338.103} C_DIS
LIN {X -0.061,Y -625.092,Z 926.673,A 0.000,B 0.000,C 90.000,E1 337.050} C_DIS
LIN {X -0.291,Y -627.989,Z 926.668,A 0.000,B 0.000,C 90.000,E1 336.305} C_DIS
LIN {X -0.211,Y -631.557,Z 926.663,A 0.000,B 0.000,C 90.000,E1 335.281} C_DIS
LIN {X -0.260,Y -636.534,Z 926.654,A 0.000,B 0.000,C 90.000,E1 333.768} C_DIS
LIN {X -0.109,Y -638.921,Z 926.650,A 0.000,B 0.000,C 90.000,E1 332.999} C_DIS
LIN {X -0.310,Y -643.142,Z 926.642,A 0.000,B 0.000,C 90.000,E1 331.513} C_DIS
LIN {X 0.213,Y -645.043,Z 926.637,A 0.000,B 0.000,C 90.000,E1 330.717} C_DIS
LIN {X -0.112,Y -648.691,Z 926.629,A 0.000,B 0.000,C 90.000,E1 329.253} C_DIS
LIN {X 0.092,Y -651.404,Z 926.622,A 0.000,B 0.000,C 90.000,E1 327.995} C_DIS
LIN {X 0.133,Y -653.638,Z 926.615,A 0.000,B 0.000,C 90.000,E1 326.755} C_DIS
LIN {X -0.242,Y -655.181,Z 926.610,A 0.000,B 0.000,C 90.000,E1 325.801} C_DIS
LIN {X -0.146,Y -656.815,Z 926.603,A 0.000,B 0.000,C 90.000,E1 324.562} C_DIS
LIN {X -0.118,Y -657.931,Z 926.598,A 0.000,B 0.000,C 90.000,E1 323.577} C_DIS
LIN {X -0.133,Y -659.211,Z 926.591,A 0.000,B 0.000,C 90.000,E1 322.351} C_DIS
LIN {X -0.201,Y -660.604,Z 926.581,A 0.000,B 0.000,C 90.000,E1 320.642} C_DIS
LIN {X -0.255,Y -662.173,Z 926.570,A 0.000,B 0.000,C 90.000,E1 318.690} C_DIS
LIN {X 0.173,Y -663.793,Z 926.561,A 0.000,B 0.000,C 90.000,E1 316.944} C_DIS
LIN {X 0.135,Y -664.685,Z 926.556,A 0.000,B 0.000,C 90.000,E1 315.972} C_DIS
LIN {X 0.097,Y -667.062,Z 926.539,A 0.000,B 0.000,C 90.000,E1 313.056} C_DIS
LIN {X 0.139,Y -668.497,Z 926.531,A 0.000,B 0.000,C 90.000,E1 311.595} C_DIS
LIN {X -0.227,Y -669.819,Z 926.523,A 0.000,B 0.000,C 90.000,E1 310.172} C_DIS
LIN {X -0.141,Y -670.667,Z 926.518,A 0.000,B 0.000,C 90.000,E1 309.197} C_DIS
LIN {X -0.050,Y -671.444,Z 926.512,A 0.000,B 0.000,C 90.000,E1 308.222} C_DIS
LIN {X 0.156,Y -672.285,Z 926.506,A 0.000,B 0.000,C 90.000,E1 306.996} C_DIS
LIN {X 0.387,Y -672.755,Z 926.500,A 0.000,B 0.000,C 90.000,E1 306.011} C_DIS
LIN {X -0.066,Y -673.503,Z 926.490,A 0.000,B 0.000,C 90.000,E1 304.119} C_DIS
LIN {X -0.313,Y -674.461,Z 926.479,A 0.000,B 0.000,C 90.000,E1 302.212} C_DIS
LIN {X 0.213,Y -675.876,Z 926.467,A 0.000,B 0.000,C 90.000,E1 300.001} C_DIS
LIN {X -0.114,Y -679.834,Z 926.448,A 0.000,B 0.000,C 90.000,E1 296.668} C_DIS
LIN {X 0.183,Y -682.064,Z 926.440,A 0.000,B 0.000,C 90.000,E1 295.207} C_DIS
LIN {X 0.032,Y -683.738,Z 926.434,A 0.000,B 0.000,C 90.000,E1 294.027} C_DIS
LIN {X -0.237,Y -684.538,Z 926.430,A 0.000,B 0.000,C 90.000,E1 293.334} C_DIS
LIN {X -0.026,Y -684.734,Z 926.428,A 0.000,B 0.000,C 90.000,E1 293.078} C_DIS
LIN {X 0.130,Y -684.796,Z 926.426,A 0.000,B 0.000,C 90.000,E1 292.589} C_DIS
LIN {X 0.340,Y -684.663,Z 926.424,A 0.000,B 0.000,C 90.000,E1 292.333} C_DIS
LIN {X -0.343,Y -684.043,Z 926.423,A 0.000,B 0.000,C 90.000,E1 292.153} C_DIS
LIN {X -0.136,Y -683.596,Z 926.422,A 0.000,B 0.000,C 90.000,E1 291.897} C_DIS
LIN {X -0.185,Y -682.737,Z 926.420,A 0.000,B 0.000,C 90.000,E1 291.663} C_DIS
LIN {X -0.083,Y -681.908,Z 926.420,A 0.000,B 0.000,C 90.000,E1 291.535} C_DIS
LIN {X 0.125,Y -677.011,Z 926.417,A 0.000,B 0.000,C 90.000,E1 291.046} C_DIS
LIN {X 0.246,Y -675.525,Z 926.416,A 0.000,B 0.000,C 90.000,E1 290.918} C_DIS
LIN {X 0.095,Y -663.319,Z 926.413,A 0.000,B 0.000,C 90.000,E1 290.248} C_DIS
LIN {X 0.040,Y -661.989,Z 926.412,A 0.000,B 0.000,C 90.000,E1 290.120} C_DIS
LIN {X -0.003,Y -661.971,Z 926.412,A 0.000,B 0.000,C 90.000,E1 290.120} C_DIS
LIN {X -0.291,Y -661.812,Z 926.411,A 0.000,B 0.000,C 90.000,E1 289.939} C_DIS
LIN {X -0.257,Y -662.417,Z 926.409,A 0.000,B 0.000,C 90.000,E1 289.631} C_DIS
LIN {X 0.107,Y -663.398,Z 926.407,A 0.000,B 0.000,C 90.000,E1 289.322} C_DIS
LIN {X 0.005,Y -664.374,Z 926.406,A 0.000,B 0.000,C 90.000,E1 289.087} C_DIS
LIN {X 0.034,Y -671.781,Z 926.398,A 0.000,B 0.000,C 90.000,E1 287.638} C_DIS
LIN {X -0.102,Y -674.121,Z 926.395,A 0.000,B 0.000,C 90.000,E1 287.166} C_DIS
LIN {X -0.080,Y -677.158,Z 926.391,A 0.000,B 0.000,C 90.000,E1 286.441} C_DIS
LIN {X -0.036,Y -679.589,Z 926.387,A 0.000,B 0.000,C 90.000,E1 285.717} C_DIS
LIN {X -0.156,Y -681.442,Z 926.383,A 0.000,B 0.000,C 90.000,E1 285.009} C_DIS
LIN {X -0.254,Y -683.053,Z 926.379,A 0.000,B 0.000,C 90.000,E1 284.300} C_DIS
LIN {X -0.335,Y -684.409,Z 926.375,A 0.000,B 0.000,C 90.000,E1 283.592} C_DIS
LIN {X 0.263,Y -685.554,Z 926.371,A 0.000,B 0.000,C 90.000,E1 282.827} C_DIS
LIN {X 0.202,Y -686.460,Z 926.367,A 0.000,B 0.000,C 90.000,E1 282.119} C_DIS
LIN {X 0.006,Y -687.082,Z 926.364,A 0.000,B 0.000,C 90.000,E1 281.422} C_DIS
LIN {X -0.012,Y -687.215,Z 926.362,A 0.000,B 0.000,C 90.000,E1 281.186} C_DIS
LIN {X -0.049,Y -687.202,Z 926.360,A 0.000,B 0.000,C 90.000,E1 280.715} C_DIS
LIN {X -0.213,Y -686.889,Z 926.357,A 0.000,B 0.000,C 90.000,E1 280.254} C_DIS
LIN {X -0.235,Y -686.581,Z 926.356,A 0.000,B 0.000,C 90.000,E1 280.018} C_DIS
LIN {X 0.279,Y -685.692,Z 926.353,A 0.000,B 0.000,C 90.000,E1 279.500} C_DIS
LIN {X 0.223,Y -684.290,Z 926.350,A 0.000,B 0.000,C 90.000,E1 279.029} C_DIS
LIN {X 0.049,Y -682.459,Z 926.348,A 0.000,B 0.000,C 90.000,E1 278.568} C_DIS
LIN {X -0.090,Y -681.430,Z 926.346,A 0.000,B 0.000,C 90.000,E1 278.341} C_DIS
LIN {X 0.290,Y -676.696,Z 926.341,A 0.000,B 0.000,C 90.000,E1 277.352} C_DIS
LIN {X -0.083,Y -672.850,Z 926.337,A 0.000,B 0.000,C 90.000,E1 276.663} C_DIS
LIN {X 0.261,Y -669.386,Z 926.334,A 0.000,B 0.000,C 90.000,E1 276.030} C_DIS
LIN {X 0.166,Y -667.906,Z 926.332,A 0.000,B 0.000,C 90.000,E1 275.796} C_DIS
LIN {X -0.196,Y -663.597,Z 926.329,A 0.000,B 0.000,C 90.000,E1 275.220} C_DIS
LIN {X 0.160,Y -659.845,Z 926.326,A 0.000,B 0.000,C 90.000,E1 274.702} C_DIS
LIN {X -0.315,Y -654.629,Z 926.323,A 0.000,B 0.000,C 90.000,E1 274.131} C_DIS
LIN {X -0.022,Y -650.120,Z 926.320,A 0.000,B 0.000,C 90.000,E1 273.612} C_DIS
LIN {X 0.311,Y -645.236,Z 926.317,A 0.000,B 0.000,C 90.000,E1 273.094} C_DIS
LIN {X 0.128,Y -638.651,Z 926.314,A 0.000,B 0.000,C 90.000,E1 272.522} C_DIS
LIN {X -0.212,Y -631.780,Z 926.311,A 0.000,B 0.000,C 90.000,E1 272.007} C_DIS
LIN {X -0.261,Y -624.321,Z 926.308,A 0.000,B 0.000,C 90.000,E1 271.489} C_DIS
LIN {X 0.017,Y -616.412,Z 926.305,A 0.000,B 0.000,C 90.000,E1 270.974} C_DIS
LIN {X 0.088,Y -611.735,Z 926.304,A 0.000,B 0.000,C 90.000,E1 270.688} C_DIS
LIN {X 0.299,Y -603.328,Z 926.301,A 0.000,B 0.000,C 90.000,E1 270.229} C_DIS
LIN {X 0.165,Y -598.302,Z 926.300,A 0.000,B 0.000,C 90.000,E1 270.000} C_DIS
LIN {X 0.037,Y -591.149,Z 926.298,A 0.000,B 0.000,C 90.000,E1 269.714} C_DIS
LIN {X 0.255,Y -583.698,Z 926.297,A 0.000,B 0.000,C 90.000,E1 269.427} C_DIS
LIN {X -0.284,Y -577.979,Z 926.296,A 0.000,B 0.000,C 90.000,E1 269.312} C_DIS
LIN {X 0.064,Y -572.187,Z 926.295,A 0.000,B 0.000,C 90.000,E1 269.141} C_DIS
LIN {X 0.041,Y -565.881,Z 926.295,A 0.000,B 0.000,C 90.000,E1 269.026} C_DIS
LIN {X 0.005,Y -560.895,Z 926.294,A 0.000,B 0.000,C 90.000,E1 268.969} C_DIS
LIN {X -0.124,Y -552.510,Z 926.294,A 0.000,B 0.000,C 90.000,E1 268.912} C_DIS
LIN {X -0.081,Y -550.792,Z 926.294,A 0.000,B 0.000,C 90.000,E1 268.854} C_DIS
LIN {X -0.113,Y -550.739,Z 926.294,A 0.000,B 0.000,C 90.000,E1 268.854} C_DIS
LIN {X 0.122,Y -549.299,Z 926.292,A 0.000,B 0.000,C 90.000,E1 268.625} C_DIS
LIN {X -0.072,Y -545.697,Z 926.290,A 0.000,B 0.000,C 90.000,E1 268.224} C_DIS
LIN {X 0.240,Y -544.167,Z 926.289,A 0.000,B 0.000,C 90.000,E1 268.051} C_DIS
LIN {X 0.198,Y -544.139,Z 926.289,A 0.000,B 0.000,C 90.000,E1 268.051} C_DIS
LIN {X -0.266,Y -543.462,Z 926.288,A 0.000,B 0.000,C 90.000,E1 267.822} C_DIS
LIN {X -0.055,Y -540.050,Z 926.267,A 0.000,B 0.000,C 90.000,E1 263.970} C_DIS
LIN {X 0.072,Y -539.082,Z 926.259,A 0.000,B 0.000,C 90.000,E1 262.534} C_DIS
LIN {X -0.216,Y -538.032,Z 926.251,A 0.000,B 0.000,C 90.000,E1 261.141} C_DIS
LIN {X -0.050,Y -537.026,Z 926.244,A 0.000,B 0.000,C 90.000,E1 259.982} C_DIS
LIN {X 0.133,Y -535.973,Z 926.240,A 0.000,B 0.000,C 90.000,E1 259.106} C_DIS
LIN {X 0.084,Y -532.554,Z 926.225,A 0.000,B 0.000,C 90.000,E1 256.533} C_DIS
LIN {X 0.065,Y -530.422,Z 926.216,A 0.000,B 0.000,C 90.000,E1 254.810} C_DIS
LIN {X 0.004,Y -528.336,Z 926.206,A 0.000,B 0.000,C 90.000,E1 253.087} C_DIS
LIN {X 0.039,Y -526.545,Z 926.198,A 0.000,B 0.000,C 90.000,E1 251.638} C_DIS
LIN {X -0.139,Y -523.535,Z 926.185,A 0.000,B 0.000,C 90.000,E1 249.337} C_DIS
LIN {X -0.153,Y -521.236,Z 926.175,A 0.000,B 0.000,C 90.000,E1 247.592} C_DIS
LIN {X 0.125,Y -519.195,Z 926.167,A 0.000,B 0.000,C 90.000,E1 246.102} C_DIS
LIN {X 0.009,Y -516.425,Z 926.158,A 0.000,B 0.000,C 90.000,E1 244.357} C_DIS
LIN {X 0.154,Y -514.148,Z 926.149,A 0.000,B 0.000,C 90.000,E1 242.871} C_DIS
LIN {X -0.190,Y -511.686,Z 926.141,A 0.000,B 0.000,C 90.000,E1 241.435} C_DIS
LIN {X 0.121,Y -509.076,Z 926.133,A 0.000,B 0.000,C 90.000,E1 239.921} C_DIS
LIN {X 0.050,Y -506.925,Z 926.126,A 0.000,B 0.000,C 90.000,E1 238.742} C_DIS
LIN {X -0.114,Y -505.203,Z 926.121,A 0.000,B 0.000,C 90.000,E1 237.867} C_DIS
LIN {X 0.284,Y -502.689,Z 926.115,A 0.000,B 0.000,C 90.000,E1 236.628} C_DIS
LIN {X -0.053,Y -499.904,Z 926.108,A 0.000,B 0.000,C 90.000,E1 235.468} C_DIS
LIN {X 0.281,Y -495.913,Z 926.098,A 0.000,B 0.000,C 90.000,E1 233.623} C_DIS
LIN {X 0.131,Y -491.977,Z 926.088,A 0.000,B 0.000,C 90.000,E1 231.823} C_DIS
LIN {X -0.172,Y -489.235,Z 926.081,A 0.000,B 0.000,C 90.000,E1 230.642} C_DIS
LIN {X 0.141,Y -485.115,Z 926.071,A 0.000,B 0.000,C 90.000,E1 228.771} C_DIS
LIN {X 0.181,Y -481.626,Z 926.063,A 0.000,B 0.000,C 90.000,E1 227.229} C_DIS
LIN {X -0.077,Y -477.514,Z 926.052,A 0.000,B 0.000,C 90.000,E1 225.405} C_DIS
LIN {X -0.301,Y -474.825,Z 926.045,A 0.000,B 0.000,C 90.000,E1 224.190} C_DIS
LIN {X -0.044,Y -470.652,Z 926.035,A 0.000,B 0.000,C 90.000,E1 222.285} C_DIS
LIN {X 0.003,Y -467.845,Z 926.028,A 0.000,B 0.000,C 90.000,E1 221.024} C_DIS
LIN {X 0.283,Y -462.423,Z 926.014,A 0.000,B 0.000,C 90.000,E1 218.463} C_DIS
LIN {X -0.076,Y -459.734,Z 926.007,A 0.000,B 0.000,C 90.000,E1 217.237} C_DIS
LIN {X -0.001,Y -455.587,Z 925.996,A 0.000,B 0.000,C 90.000,E1 215.311} C_DIS
LIN {X -0.007,Y -452.089,Z 925.987,A 0.000,B 0.000,C 90.000,E1 213.706} C_DIS
LIN {X -0.178,Y -447.089,Z 925.975,A 0.000,B 0.000,C 90.000,E1 211.465} C_DIS
LIN {X -0.004,Y -442.760,Z 925.964,A 0.000,B 0.000,C 90.000,E1 209.489} C_DIS
LIN {X -0.011,Y -439.984,Z 925.957,A 0.000,B 0.000,C 90.000,E1 208.180} C_DIS
LIN {X -0.214,Y -435.644,Z 925.946,A 0.000,B 0.000,C 90.000,E1 206.232} C_DIS
LIN {X -0.135,Y -429.800,Z 925.931,A 0.000,B 0.000,C 90.000,E1 203.567} C_DIS
LIN {X -0.146,Y -426.141,Z 925.922,A 0.000,B 0.000,C 90.000,E1 201.897} C_DIS
LIN {X -0.169,Y -423.207,Z 925.914,A 0.000,B 0.000,C 90.000,E1 200.556} C_DIS
LIN {X 0.214,Y -417.065,Z 925.897,A 0.000,B 0.000,C 90.000,E1 197.457} C_DIS
LIN {X 0.161,Y -415.039,Z 925.892,A 0.000,B 0.000,C 90.000,E1 196.441} C_DIS
LIN {X -0.149,Y -411.528,Z 925.882,A 0.000,B 0.000,C 90.000,E1 194.773} C_DIS
LIN {X 0.166,Y -408.032,Z 925.872,A 0.000,B 0.000,C 90.000,E1 193.008} C_DIS
LIN {X 0.013,Y -403.885,Z 925.861,A 0.000,B 0.000,C 90.000,E1 190.950} C_DIS
LIN {X 0.002,Y -399.790,Z 925.849,A 0.000,B 0.000,C 90.000,E1 188.859} C_DIS
LIN {X -0.042,Y -397.699,Z 925.843,A 0.000,B 0.000,C 90.000,E1 187.814} C_DIS
LIN {X 0.119,Y -394.271,Z 925.834,A 0.000,B 0.000,C 90.000,E1 186.030} C_DIS
LIN {X -0.087,Y -388.447,Z 925.816,A 0.000,B 0.000,C 90.000,E1 182.865} C_DIS
LIN {X -0.149,Y -381.648,Z 925.792,A 0.000,B 0.000,C 90.000,E1 178.568} C_DIS
LIN {X 0.041,Y -379.847,Z 925.782,A 0.000,B 0.000,C 90.000,E1 176.731} C_DIS
LIN {X 0.163,Y -379.623,Z 925.778,A 0.000,B 0.000,C 90.000,E1 175.988} C_DIS
LIN {X -0.073,Y -379.881,Z 925.774,A 0.000,B 0.000,C 90.000,E1 175.298} C_DIS
LIN {X -0.140,Y -380.370,Z 925.772,A 0.000,B 0.000,C 90.000,E1 174.951} C_DIS
LIN {X 0.075,Y -381.457,Z 925.769,A 0.000,B 0.000,C 90.000,E1 174.375} C_DIS
LIN {X 0.008,Y -381.971,Z 925.768,A 0.000,B 0.000,C 90.000,E1 174.204} C_DIS
LIN {X -0.095,Y -384.286,Z 925.765,A 0.000,B 0.000,C 90.000,E1 173.628} C_DIS
LIN {X 0.034,Y -385.859,Z 925.763,A 0.000,B 0.000,C 90.000,E1 173.337} C_DIS
LIN {X -0.181,Y -387.932,Z 925.761,A 0.000,B 0.000,C 90.000,E1 173.053} C_DIS
LIN {X -0.022,Y -390.484,Z 925.760,A 0.000,B 0.000,C 90.000,E1 172.704} C_DIS
LIN {X 0.032,Y -395.139,Z 925.757,A 0.000,B 0.000,C 90.000,E1 172.243} C_DIS
LIN {X -0.103,Y -399.583,Z 925.755,A 0.000,B 0.000,C 90.000,E1 171.894} C_DIS
LIN {X 0.121,Y -406.287,Z 925.752,A 0.000,B 0.000,C 90.000,E1 171.376} C_DIS
LIN {X 0.173,Y -412.690,Z 925.750,A 0.000,B 0.000,C 90.000,E1 170.905} C_DIS
LIN {X -0.066,Y -425.616,Z 925.744,A 0.000,B 0.000,C 90.000,E1 169.982} C_DIS
LIN {X 0.117,Y -435.067,Z 925.740,A 0.000,B 0.000,C 90.000,E1 169.218} C_DIS
LIN {X -0.143,Y -445.679,Z 925.735,A 0.000,B 0.000,C 90.000,E1 168.342} C_DIS
LIN {X -0.174,Y -451.658,Z 925.732,A 0.000,B 0.000,C 90.000,E1 167.813} C_DIS
LIN {X -0.052,Y -461.941,Z 925.727,A 0.000,B 0.000,C 90.000,E1 166.825} C_DIS
LIN {X -0.081,Y -468.766,Z 925.723,A 0.000,B 0.000,C 90.000,E1 166.117} C_DIS
LIN {X -0.162,Y -476.726,Z 925.718,A 0.000,B 0.000,C 90.000,E1 165.227} C_DIS
LIN {X -0.084,Y -485.797,Z 925.712,A 0.000,B 0.000,C 90.000,E1 164.157} C_DIS
LIN {X 0.028,Y -491.843,Z 925.708,A 0.000,B 0.000,C 90.000,E1 163.378} C_DIS
LIN {X -0.163,Y -498.779,Z 925.703,A 0.000,B 0.000,C 90.000,E1 162.489} C_DIS
LIN {X -0.322,Y -510.413,Z 925.693,A 0.000,B 0.000,C 90.000,E1 160.859} C_DIS
LIN {X 0.167,Y -520.285,Z 925.685,A 0.000,B 0.000,C 90.000,E1 159.337} C_DIS
LIN {X 0.307,Y -527.820,Z 925.679,A 0.000,B 0.000,C 90.000,E1 158.156} C_DIS
LIN {X 0.166,Y -533.275,Z 925.674,A 0.000,B 0.000,C 90.000,E1 157.305} C_DIS
LIN {X -0.037,Y -543.803,Z 925.665,A 0.000,B 0.000,C 90.000,E1 155.613} C_DIS
LIN {X 0.307,Y -549.640,Z 925.659,A 0.000,B 0.000,C 90.000,E1 154.588} C_DIS
LIN {X -0.117,Y -556.012,Z 925.653,A 0.000,B 0.000,C 90.000,E1 153.512} C_DIS
LIN {X -0.006,Y -560.398,Z 925.648,A 0.000,B 0.000,C 90.000,E1 152.666} C_DIS
LIN {X -0.108,Y -564.745,Z 925.644,A 0.000,B 0.000,C 90.000,E1 151.847} C_DIS
LIN {X -0.070,Y -572.099,Z 925.635,A 0.000,B 0.000,C 90.000,E1 150.333} C_DIS
LIN {X -0.284,Y -575.844,Z 925.631,A 0.000,B 0.000,C 90.000,E1 149.537} C_DIS
LIN {X 0.178,Y -580.562,Z 925.625,A 0.000,B 0.000,C 90.000,E1 148.408} C_DIS
LIN {X 0.209,Y -585.020,Z 925.619,A 0.000,B 0.000,C 90.000,E1 147.327} C_DIS
LIN {X 0.002,Y -590.542,Z 925.611,A 0.000,B 0.000,C 90.000,E1 146.008} C_DIS
LIN {X -0.326,Y -594.862,Z 925.605,A 0.000,B 0.000,C 90.000,E1 144.975} C_DIS
LIN {X -0.256,Y -598.853,Z 925.599,A 0.000,B 0.000,C 90.000,E1 143.909} C_DIS
LIN {X -0.101,Y -604.654,Z 925.591,A 0.000,B 0.000,C 90.000,E1 142.316} C_DIS
LIN {X -0.014,Y -611.646,Z 925.581,A 0.000,B 0.000,C 90.000,E1 140.481} C_DIS
LIN {X 0.096,Y -616.713,Z 925.573,A 0.000,B 0.000,C 90.000,E1 139.175} C_DIS
LIN {X -0.244,Y -621.691,Z 925.566,A 0.000,B 0.000,C 90.000,E1 137.919} C_DIS
LIN {X -0.221,Y -624.750,Z 925.562,A 0.000,B 0.000,C 90.000,E1 137.148} C_DIS
LIN {X -0.298,Y -628.968,Z 925.556,A 0.000,B 0.000,C 90.000,E1 136.134} C_DIS
LIN {X 0.121,Y -633.049,Z 925.551,A 0.000,B 0.000,C 90.000,E1 135.081} C_DIS
LIN {X -0.401,Y -638.086,Z 925.544,A 0.000,B 0.000,C 90.000,E1 133.866} C_DIS
LIN {X -0.383,Y -642.981,Z 925.537,A 0.000,B 0.000,C 90.000,E1 132.609} C_DIS
LIN {X 0.061,Y -649.840,Z 925.527,A 0.000,B 0.000,C 90.000,E1 130.825} C_DIS
LIN {X 0.334,Y -654.625,Z 925.520,A 0.000,B 0.000,C 90.000,E1 129.564} C_DIS
LIN {X -0.213,Y -661.241,Z 925.510,A 0.000,B 0.000,C 90.000,E1 127.890} C_DIS
LIN {X -0.083,Y -667.612,Z 925.501,A 0.000,B 0.000,C 90.000,E1 126.171} C_DIS
LIN {X 0.070,Y -671.924,Z 925.494,A 0.000,B 0.000,C 90.000,E1 124.945} C_DIS
LIN {X 0.455,Y -675.992,Z 925.488,A 0.000,B 0.000,C 90.000,E1 123.706} C_DIS
LIN {X -0.178,Y -678.200,Z 925.484,A 0.000,B 0.000,C 90.000,E1 123.038} C_DIS
LIN {X 0.311,Y -681.344,Z 925.477,A 0.000,B 0.000,C 90.000,E1 121.799} C_DIS
LIN {X 0.116,Y -682.509,Z 925.474,A 0.000,B 0.000,C 90.000,E1 121.337} C_DIS
LIN {X 0.100,Y -684.563,Z 925.469,A 0.000,B 0.000,C 90.000,E1 120.384} C_DIS
LIN {X 0.140,Y -685.952,Z 925.465,A 0.000,B 0.000,C 90.000,E1 119.667} C_DIS
LIN {X 0.196,Y -687.208,Z 925.461,A 0.000,B 0.000,C 90.000,E1 118.949} C_DIS
LIN {X 0.266,Y -688.305,Z 925.457,A 0.000,B 0.000,C 90.000,E1 118.231} C_DIS
LIN {X -0.036,Y -689.356,Z 925.452,A 0.000,B 0.000,C 90.000,E1 117.308} C_DIS
LIN {X 0.204,Y -689.967,Z 925.445,A 0.000,B 0.000,C 90.000,E1 116.104} C_DIS
LIN {X -0.009,Y -690.060,Z 925.441,A 0.000,B 0.000,C 90.000,E1 115.412} C_DIS
LIN {X 0.070,Y -690.098,Z 925.437,A 0.000,B 0.000,C 90.000,E1 114.695} C_DIS
LIN {X -0.146,Y -689.849,Z 925.433,A 0.000,B 0.000,C 90.000,E1 114.003} C_DIS
LIN {X 0.039,Y -689.458,Z 925.431,A 0.000,B 0.000,C 90.000,E1 113.515} C_DIS
LIN {X 0.225,Y -688.279,Z 925.428,A 0.000,B 0.000,C 90.000,E1 113.025} C_DIS
LIN {X -0.183,Y -687.566,Z 925.427,A 0.000,B 0.000,C 90.000,E1 112.823} C_DIS
LIN {X -0.072,Y -686.909,Z 925.426,A 0.000,B 0.000,C 90.000,E1 112.695} C_DIS
LIN {X 0.097,Y -683.532,Z 925.423,A 0.000,B 0.000,C 90.000,E1 112.206} C_DIS
LIN {X 0.200,Y -682.431,Z 925.423,A 0.000,B 0.000,C 90.000,E1 112.078} C_DIS
LIN {X 0.046,Y -680.738,Z 925.422,A 0.000,B 0.000,C 90.000,E1 111.972} C_DIS
LIN {X 0.148,Y -677.947,Z 925.421,A 0.000,B 0.000,C 90.000,E1 111.844} C_DIS
LIN {X -0.005,Y -673.747,Z 925.421,A 0.000,B 0.000,C 90.000,E1 111.716} C_DIS
LIN {X 0.149,Y -671.096,Z 925.420,A 0.000,B 0.000,C 90.000,E1 111.589} C_DIS
LIN {X -0.059,Y -668.768,Z 925.420,A 0.000,B 0.000,C 90.000,E1 111.535} C_DIS
LIN {X -0.020,Y -663.426,Z 925.419,A 0.000,B 0.000,C 90.000,E1 111.461} C_DIS
LIN {X 0.205,Y -658.557,Z 925.419,A 0.000,B 0.000,C 90.000,E1 111.408} C_DIS
LIN {X 0.139,Y -652.607,Z 925.419,A 0.000,B 0.000,C 90.000,E1 111.408} C_DIS
LIN {X 0.074,Y -643.831,Z 925.419,A 0.000,B 0.000,C 90.000,E1 111.408} C_DIS
LIN {X -0.026,Y -640.754,Z 925.419,A 0.000,B 0.000,C 90.000,E1 111.408} C_DIS
LIN {X 0.054,Y -635.763,Z 925.419,A 0.000,B 0.000,C 90.000,E1 111.354} C_DIS
LIN {X -0.173,Y -629.409,Z 925.418,A 0.000,B 0.000,C 90.000,E1 111.280} C_DIS
LIN {X -0.022,Y -623.759,Z 925.418,A 0.000,B 0.000,C 90.000,E1 111.153} C_DIS
LIN {X -0.312,Y -620.350,Z 925.417,A 0.000,B 0.000,C 90.000,E1 111.099} C_DIS
LIN {X -0.133,Y -614.754,Z 925.416,A 0.000,B 0.000,C 90.000,E1 110.918} C_DIS
LIN {X 0.176,Y -606.354,Z 925.414,A 0.000,B 0.000,C 90.000,E1 110.556} C_DIS
LIN {X 0.111,Y -603.472,Z 925.414,A 0.000,B 0.000,C 90.000,E1 110.429} C_DIS
LIN {X -0.161,Y -598.242,Z 925.412,A 0.000,B 0.000,C 90.000,E1 110.174} C_DIS
LIN {X 0.175,Y -588.613,Z 925.409,A 0.000,B 0.000,C 90.000,E1 109.523} C_DIS
LIN {X 0.076,Y -581.330,Z 925.406,A 0.000,B 0.000,C 90.000,E1 109.033} C_DIS
LIN {X -0.142,Y -578.230,Z 925.405,A 0.000,B 0.000,C 90.000,E1 108.852} C_DIS
LIN {X -0.072,Y -571.325,Z 925.403,A 0.000,B 0.000,C 90.000,E1 108.471} C_DIS
LIN {X -0.257,Y -564.458,Z 925.401,A 0.000,B 0.000,C 90.000,E1 108.181} C_DIS
LIN {X -0.019,Y -557.407,Z 925.399,A 0.000,B 0.000,C 90.000,E1 107.873} C_DIS
LIN {X -0.165,Y -554.632,Z 925.399,A 0.000,B 0.000,C 90.000,E1 107.747} C_DIS
LIN {X 0.015,Y -553.077,Z 925.398,A 0.000,B 0.000,C 90.000,E1 107.583} C_DIS
LIN {X -0.019,Y -553.063,Z 925.398,A 0.000,B 0.000,C 90.000,E1 107.583} C_DIS
LIN {X -0.218,Y -552.669,Z 925.397,A 0.000,B 0.000,C 90.000,E1 107.402} C_DIS
LIN {X -0.103,Y -552.858,Z 925.392,A 0.000,B 0.000,C 90.000,E1 106.551} C_DIS
LIN {X 0.081,Y -553.494,Z 925.384,A 0.000,B 0.000,C 90.000,E1 105.134} C_DIS
LIN {X 0.252,Y -554.600,Z 925.372,A 0.000,B 0.000,C 90.000,E1 102.883} C_DIS
LIN {X -0.217,Y -556.300,Z 925.358,A 0.000,B 0.000,C 90.000,E1 100.423} C_DIS
LIN {X -0.194,Y -557.414,Z 925.350,A 0.000,B 0.000,C 90.000,E1 99.029} C_DIS
LIN {X -0.096,Y -558.630,Z 925.341,A 0.000,B 0.000,C 90.000,E1 97.352} C_DIS
LIN {X -0.245,Y -559.389,Z 925.335,A 0.000,B 0.000,C 90.000,E1 96.258} C_DIS
LIN {X -0.169,Y -560.415,Z 925.325,A 0.000,B 0.000,C 90.000,E1 94.588} C_DIS
LIN {X -0.029,Y -561.420,Z 925.315,A 0.000,B 0.000,C 90.000,E1 92.636} C_DIS
LIN {X -0.087,Y -561.996,Z 925.307,A 0.000,B 0.000,C 90.000,E1 91.260} C_DIS
LIN {X -0.249,Y -562.417,Z 925.301,A 0.000,B 0.000,C 90.000,E1 90.172} C_DIS
LIN {X 0.261,Y -562.753,Z 925.293,A 0.000,B 0.000,C 90.000,E1 88.740} C_DIS
LIN {X -0.236,Y -563.100,Z 925.284,A 0.000,B 0.000,C 90.000,E1 87.135} C_DIS
LIN {X -0.232,Y -563.351,Z 925.276,A 0.000,B 0.000,C 90.000,E1 85.755} C_DIS
LIN {X -0.125,Y -563.601,Z 925.267,A 0.000,B 0.000,C 90.000,E1 84.090} C_DIS
LIN {X 0.103,Y -563.931,Z 925.258,A 0.000,B 0.000,C 90.000,E1 82.413} C_DIS
LIN {X 0.116,Y -564.540,Z 925.246,A 0.000,B 0.000,C 90.000,E1 80.208} C_DIS
LIN {X 0.074,Y -565.371,Z 925.235,A 0.000,B 0.000,C 90.000,E1 78.285} C_DIS
LIN {X -0.013,Y -566.307,Z 925.226,A 0.000,B 0.000,C 90.000,E1 76.645} C_DIS
LIN {X -0.124,Y -567.154,Z 925.218,A 0.000,B 0.000,C 90.000,E1 75.283} C_DIS
LIN {X -0.221,Y -567.935,Z 925.211,A 0.000,B 0.000,C 90.000,E1 73.921} C_DIS
LIN {X 0.185,Y -568.727,Z 925.201,A 0.000,B 0.000,C 90.000,E1 72.236} C_DIS
LIN {X -0.310,Y -569.538,Z 925.191,A 0.000,B 0.000,C 90.000,E1 70.369} C_DIS
LIN {X -0.188,Y -569.850,Z 925.185,A 0.000,B 0.000,C 90.000,E1 69.263} C_DIS
LIN {X -0.056,Y -570.239,Z 925.179,A 0.000,B 0.000,C 90.000,E1 68.156} C_DIS
LIN {X 0.252,Y -570.499,Z 925.170,A 0.000,B 0.000,C 90.000,E1 66.485} C_DIS
LIN {X 0.269,Y -570.723,Z 925.160,A 0.000,B 0.000,C 90.000,E1 64.845} C_DIS
LIN {X -0.225,Y -570.904,Z 925.151,A 0.000,B 0.000,C 90.000,E1 63.256} C_DIS
LIN {X 0.040,Y -570.886,Z 925.142,A 0.000,B 0.000,C 90.000,E1 61.591} C_DIS
LIN {X 0.066,Y -570.888,Z 925.133,A 0.000,B 0.000,C 90.000,E1 59.950} C_DIS
LIN {X -0.108,Y -570.723,Z 925.124,A 0.000,B 0.000,C 90.000,E1 58.329} C_DIS
LIN {X -0.096,Y -570.237,Z 925.116,A 0.000,B 0.000,C 90.000,E1 56.962} C_DIS
LIN {X -0.221,Y -569.747,Z 925.110,A 0.000,B 0.000,C 90.000,E1 55.881} C_DIS
LIN {X -0.163,Y -569.273,Z 925.106,A 0.000,B 0.000,C 90.000,E1 55.055} C_DIS
LIN {X 0.215,Y -568.716,Z 925.101,A 0.000,B 0.000,C 90.000,E1 54.196} C_DIS
LIN {X -0.204,Y -568.071,Z 925.097,A 0.000,B 0.000,C 90.000,E1 53.417} C_DIS
LIN {X 0.287,Y -566.941,Z 925.091,A 0.000,B 0.000,C 90.000,E1 52.271} C_DIS
LIN {X 0.310,Y -565.643,Z 925.085,A 0.000,B 0.000,C 90.000,E1 51.170} C_DIS
LIN {X -0.119,Y -564.001,Z 925.078,A 0.000,B 0.000,C 90.000,E1 50.114} C_DIS
LIN {X 0.089,Y -563.150,Z 925.075,A 0.000,B 0.000,C 90.000,E1 49.542} C_DIS
LIN {X -0.045,Y -561.610,Z 925.071,A 0.000,B 0.000,C 90.000,E1 48.728} C_DIS
LIN {X 0.171,Y -559.900,Z 925.066,A 0.000,B 0.000,C 90.000,E1 47.877} C_DIS
LIN {X -0.039,Y -557.936,Z 925.062,A 0.000,B 0.000,C 90.000,E1 47.067} C_DIS
LIN {X 0.140,Y -555.689,Z 925.057,A 0.000,B 0.000,C 90.000,E1 46.215} C_DIS
LIN {X 0.241,Y -554.102,Z 925.054,A 0.000,B 0.000,C 90.000,E1 45.648} C_DIS
LIN {X -0.021,Y -551.344,Z 925.049,A 0.000,B 0.000,C 90.000,E1 44.838} C_DIS
LIN {X 0.049,Y -549.389,Z 925.046,A 0.000,B 0.000,C 90.000,E1 44.271} C_DIS
LIN {X -0.261,Y -546.045,Z 925.041,A 0.000,B 0.000,C 90.000,E1 43.461} C_DIS
LIN {X -0.036,Y -543.038,Z 925.037,A 0.000,B 0.000,C 90.000,E1 42.732} C_DIS
LIN {X -0.001,Y -540.392,Z 925.034,A 0.000,B 0.000,C 90.000,E1 42.162} C_DIS
LIN {X -0.021,Y -537.546,Z 925.031,A 0.000,B 0.000,C 90.000,E1 41.595} C_DIS
LIN {X -0.073,Y -532.915,Z 925.026,A 0.000,B 0.000,C 90.000,E1 40.744} C_DIS
LIN {X 0.084,Y -530.412,Z 925.024,A 0.000,B 0.000,C 90.000,E1 40.297} C_DIS
LIN {X 0.167,Y -524.178,Z 925.018,A 0.000,B 0.000,C 90.000,E1 39.277} C_DIS
LIN {X 0.042,Y -518.481,Z 925.013,A 0.000,B 0.000,C 90.000,E1 38.418} C_DIS
LIN {X 0.174,Y -512.411,Z 925.009,A 0.000,B 0.000,C 90.000,E1 37.523} C_DIS
LIN {X 0.016,Y -508.090,Z 925.005,A 0.000,B 0.000,C 90.000,E1 36.950} C_DIS
LIN {X -0.276,Y -501.138,Z 925.000,A 0.000,B 0.000,C 90.000,E1 36.091} C_DIS
LIN {X 0.184,Y -496.049,Z 924.997,A 0.000,B 0.000,C 90.000,E1 35.438} C_DIS
LIN {X -0.154,Y -489.286,Z 924.993,A 0.000,B 0.000,C 90.000,E1 34.739} C_DIS
LIN {X 0.075,Y -485.147,Z 924.991,A 0.000,B 0.000,C 90.000,E1 34.278} C_DIS
LIN {X -0.030,Y -480.862,Z 924.988,A 0.000,B 0.000,C 90.000,E1 33.865} C_DIS
LIN {X 0.159,Y -475.082,Z 924.985,A 0.000,B 0.000,C 90.000,E1 33.293} C_DIS
LIN {X 0.066,Y -466.188,Z 924.981,A 0.000,B 0.000,C 90.000,E1 32.498} C_DIS
LIN {X -0.050,Y -458.667,Z 924.977,A 0.000,B 0.000,C 90.000,E1 31.848} C_DIS
LIN {X 0.052,Y -446.377,Z 924.971,A 0.000,B 0.000,C 90.000,E1 30.797} C_DIS
LIN {X -0.163,Y -426.601,Z 924.962,A 0.000,B 0.000,C 90.000,E1 29.155} C_DIS
LIN {X 0.111,Y -411.643,Z 924.954,A 0.000,B 0.000,C 90.000,E1 27.769} C_DIS
LIN {X 0.089,Y -398.334,Z 924.947,A 0.000,B 0.000,C 90.000,E1 26.437} C_DIS
LIN {X 0.221,Y -393.777,Z 924.944,A 0.000,B 0.000,C 90.000,E1 25.848} C_DIS
LIN {X -0.087,Y -391.559,Z 924.942,A 0.000,B 0.000,C 90.000,E1 25.515} C_DIS
LIN {X 0.127,Y -389.622,Z 924.939,A 0.000,B 0.000,C 90.000,E1 24.951} C_DIS
LIN {X -0.015,Y -388.763,Z 924.935,A 0.000,B 0.000,C 90.000,E1 24.259} C_DIS
LIN {X -0.151,Y -388.762,Z 924.930,A 0.000,B 0.000,C 90.000,E1 23.387} C_DIS
LIN {X 0.016,Y -390.705,Z 924.916,A 0.000,B 0.000,C 90.000,E1 20.865} C_DIS
LIN {X 0.112,Y -393.371,Z 924.902,A 0.000,B 0.000,C 90.000,E1 18.362} C_DIS
LIN {X -0.036,Y -395.894,Z 924.890,A 0.000,B 0.000,C 90.000,E1 16.260} C_DIS
LIN {X 0.117,Y -399.065,Z 924.877,A 0.000,B 0.000,C 90.000,E1 13.772} C_DIS
LIN {X -0.138,Y -403.180,Z 924.861,A 0.000,B 0.000,C 90.000,E1 11.007} C_DIS
LIN {X -0.104,Y -407.686,Z 924.846,A 0.000,B 0.000,C 90.000,E1 8.219} C_DIS
LIN {X -0.063,Y -412.043,Z 924.832,A 0.000,B 0.000,C 90.000,E1 5.796} C_DIS
LIN {X -0.015,Y -415.374,Z 924.823,A 0.000,B 0.000,C 90.000,E1 4.073} C_DIS
LIN {X 0.133,Y -419.698,Z 924.811,A 0.000,B 0.000,C 90.000,E1 2.007} C_DIS
LIN {X 0.160,Y -424.867,Z 924.799,A 0.000,B 0.000,C 90.000,E1 359.771} C_DIS
LIN {X 0.030,Y -429.083,Z 924.790,A 0.000,B 0.000,C 90.000,E1 358.108} C_DIS
LIN {X 0.167,Y -431.302,Z 924.786,A 0.000,B 0.000,C 90.000,E1 357.421} C_DIS
LIN {X 0.015,Y -433.681,Z 924.783,A 0.000,B 0.000,C 90.000,E1 356.963} C_DIS
LIN {X 0.078,Y -434.742,Z 924.782,A 0.000,B 0.000,C 90.000,E1 356.788} C_DIS
LIN {X 0.186,Y -437.400,Z 924.780,A 0.000,B 0.000,C 90.000,E1 356.445} C_DIS
LIN {X 0.172,Y -441.131,Z 924.779,A 0.000,B 0.000,C 90.000,E1 356.159} C_DIS
LIN {X 0.112,Y -443.048,Z 924.778,A 0.000,B 0.000,C 90.000,E1 356.045} C_DIS
LIN {X 0.215,Y -447.132,Z 924.777,A 0.000,B 0.000,C 90.000,E1 355.812} C_DIS
LIN {X -0.012,Y -458.898,Z 924.774,A 0.000,B 0.000,C 90.000,E1 355.298} C_DIS
LIN {X 0.185,Y -465.654,Z 924.772,A 0.000,B 0.000,C 90.000,E1 354.951} C_DIS
LIN {X -0.096,Y -482.182,Z 924.767,A 0.000,B 0.000,C 90.000,E1 354.147} C_DIS
LIN {X -0.181,Y -495.537,Z 924.764,A 0.000,B 0.000,C 90.000,E1 353.451} C_DIS
LIN {X -0.005,Y -505.321,Z 924.760,A 0.000,B 0.000,C 90.000,E1 352.875} C_DIS
LIN {X 0.133,Y -516.412,Z 924.757,A 0.000,B 0.000,C 90.000,E1 352.186} C_DIS
LIN {X 0.154,Y -522.635,Z 924.754,A 0.000,B 0.000,C 90.000,E1 351.781} C_DIS
LIN {X 0.088,Y -530.162,Z 924.752,A 0.000,B 0.000,C 90.000,E1 351.254} C_DIS
LIN {X 0.199,Y -536.065,Z 924.749,A 0.000,B 0.000,C 90.000,E1 350.792} C_DIS
LIN {X 0.079,Y -541.758,Z 924.746,A 0.000,B 0.000,C 90.000,E1 350.330} C_DIS
LIN {X -0.104,Y -547.273,Z 924.744,A 0.000,B 0.000,C 90.000,E1 349.859} C_DIS
LIN {X -0.028,Y -552.655,Z 924.741,A 0.000,B 0.000,C 90.000,E1 349.342} C_DIS
LIN {X -0.102,Y -557.737,Z 924.738,A 0.000,B 0.000,C 90.000,E1 348.814} C_DIS
LIN {X 0.120,Y -565.982,Z 924.732,A 0.000,B 0.000,C 90.000,E1 347.825} C_DIS
LIN {X -0.221,Y -571.441,Z 924.729,A 0.000,B 0.000,C 90.000,E1 347.173} C_DIS
LIN {X 0.257,Y -578.408,Z 924.723,A 0.000,B 0.000,C 90.000,E1 346.172} C_DIS
LIN {X 0.029,Y -582.954,Z 924.720,A 0.000,B 0.000,C 90.000,E1 345.519} C_DIS
LIN {X 0.004,Y -589.703,Z 924.714,A 0.000,B 0.000,C 90.000,E1 344.448} C_DIS
LIN {X -0.165,Y -596.414,Z 924.707,A 0.000,B 0.000,C 90.000,E1 343.268} C_DIS
LIN {X 0.160,Y -601.855,Z 924.701,A 0.000,B 0.000,C 90.000,E1 342.181} C_DIS
LIN {X 0.077,Y -605.806,Z 924.697,A 0.000,B 0.000,C 90.000,E1 341.402} C_DIS
LIN {X -0.094,Y -612.062,Z 924.690,A 0.000,B 0.000,C 90.000,E1 340.115} C_DIS
LIN {X -0.110,Y -616.123,Z 924.685,A 0.000,B 0.000,C 90.000,E1 339.209} C_DIS
LIN {X -0.121,Y -621.648,Z 924.677,A 0.000,B 0.000,C 90.000,E1 337.922} C_DIS
LIN {X 0.190,Y -625.691,Z 924.672,A 0.000,B 0.000,C 90.000,E1 336.869} C_DIS
LIN {X -0.020,Y -629.428,Z 924.666,A 0.000,B 0.000,C 90.000,E1 335.869} C_DIS
LIN {X 0.083,Y -632.893,Z 924.660,A 0.000,B 0.000,C 90.000,E1 334.845} C_DIS
LIN {X 0.008,Y -637.083,Z 924.653,A 0.000,B 0.000,C 90.000,E1 333.589} C_DIS
LIN {X 0.107,Y -638.661,Z 924.651,A 0.000,B 0.000,C 90.000,E1 333.076} C_DIS
LIN {X -0.169,Y -642.240,Z 924.644,A 0.000,B 0.000,C 90.000,E1 331.847} C_DIS
LIN {X -0.148,Y -644.923,Z 924.638,A 0.000,B 0.000,C 90.000,E1 330.845} C_DIS
LIN {X -0.001,Y -647.960,Z 924.631,A 0.000,B 0.000,C 90.000,E1 329.587} C_DIS
LIN {X 0.110,Y -650.270,Z 924.626,A 0.000,B 0.000,C 90.000,E1 328.584} C_DIS
LIN {X 0.249,Y -652.344,Z 924.620,A 0.000,B 0.000,C 90.000,E1 327.582} C_DIS
LIN {X -0.142,Y -654.076,Z 924.615,A 0.000,B 0.000,C 90.000,E1 326.628} C_DIS
LIN {X 0.396,Y -655.611,Z 924.609,A 0.000,B 0.000,C 90.000,E1 325.595} C_DIS
LIN {X -0.050,Y -656.596,Z 924.605,A 0.000,B 0.000,C 90.000,E1 324.895} C_DIS
LIN {X 0.061,Y -658.071,Z 924.598,A 0.000,B 0.000,C 90.000,E1 323.657} C_DIS
LIN {X 0.047,Y -659.366,Z 924.591,A 0.000,B 0.000,C 90.000,E1 322.431} C_DIS
LIN {X -0.021,Y -660.812,Z 924.582,A 0.000,B 0.000,C 90.000,E1 320.723} C_DIS
LIN {X -0.071,Y -662.356,Z 924.571,A 0.000,B 0.000,C 90.000,E1 318.771} C_DIS
LIN {X -0.125,Y -664.023,Z 924.561,A 0.000,B 0.000,C 90.000,E1 317.067} C_DIS
LIN {X 0.325,Y -664.932,Z 924.556,A 0.000,B 0.000,C 90.000,E1 316.053} C_DIS
LIN {X 0.299,Y -666.808,Z 924.543,A 0.000,B 0.000,C 90.000,E1 313.623} C_DIS
LIN {X 0.344,Y -668.490,Z 924.533,A 0.000,B 0.000,C 90.000,E1 311.919} C_DIS
LIN {X -0.016,Y -669.814,Z 924.525,A 0.000,B 0.000,C 90.000,E1 310.496} C_DIS
LIN {X 0.077,Y -670.903,Z 924.518,A 0.000,B 0.000,C 90.000,E1 309.277} C_DIS
LIN {X -0.246,Y -671.846,Z 924.512,A 0.000,B 0.000,C 90.000,E1 308.096} C_DIS
LIN {X -0.028,Y -672.682,Z 924.505,A 0.000,B 0.000,C 90.000,E1 306.870} C_DIS
LIN {X 0.213,Y -673.090,Z 924.500,A 0.000,B 0.000,C 90.000,E1 305.884} C_DIS
LIN {X 0.183,Y -673.786,Z 924.490,A 0.000,B 0.000,C 90.000,E1 304.199} C_DIS
LIN {X 0.026,Y -674.334,Z 924.483,A 0.000,B 0.000,C 90.000,E1 303.007} C_DIS
LIN {X 0.073,Y -675.022,Z 924.477,A 0.000,B 0.000,C 90.000,E1 301.799} C_DIS
LIN {X -0.199,Y -679.396,Z 924.451,A 0.000,B 0.000,C 90.000,E1 297.257} C_DIS
LIN {X -0.111,Y -682.214,Z 924.441,A 0.000,B 0.000,C 90.000,E1 295.335} C_DIS
LIN {X 0.019,Y -683.904,Z 924.434,A 0.000,B 0.000,C 90.000,E1 294.131} C_DIS
LIN {X 0.373,Y -684.674,Z 924.430,A 0.000,B 0.000,C 90.000,E1 293.387} C_DIS
LIN {X -0.103,Y -684.983,Z 924.427,A 0.000,B 0.000,C 90.000,E1 292.950} C_DIS
LIN {X 0.055,Y -685.000,Z 924.425,A 0.000,B 0.000,C 90.000,E1 292.461} C_DIS
LIN {X 0.264,Y -684.503,Z 924.424,A 0.000,B 0.000,C 90.000,E1 292.206} C_DIS
LIN {X -0.118,Y -683.281,Z 924.421,A 0.000,B 0.000,C 90.000,E1 291.770} C_DIS
LIN {X -0.018,Y -682.731,Z 924.420,A 0.000,B 0.000,C 90.000,E1 291.642} C_DIS
LIN {X -0.168,Y -681.884,Z 924.420,A 0.000,B 0.000,C 90.000,E1 291.535} C_DIS
LIN {X -0.068,Y -680.639,Z 924.419,A 0.000,B 0.000,C 90.000,E1 291.408} C_DIS
LIN {X 0.027,Y -677.983,Z 924.418,A 0.000,B 0.000,C 90.000,E1 291.173} C_DIS
LIN {X 0.268,Y -676.901,Z 924.417,A 0.000,B 0.000,C 90.000,E1 291.046} C_DIS
LIN {X -0.247,Y -675.445,Z 924.416,A 0.000,B 0.000,C 90.000,E1 290.972} C_DIS
LIN {X -0.259,Y -665.540,Z 924.413,A 0.000,B 0.000,C 90.000,E1 290.429} C_DIS
LIN {X -0.277,Y -663.211,Z 924.413,A 0.000,B 0.000,C 90.000,E1 290.301} C_DIS
LIN {X -0.237,Y -661.950,Z 924.412,A 0.000,B 0.000,C 90.000,E1 290.174} C_DIS
LIN {X 0.322,Y -661.920,Z 924.412,A 0.000,B 0.000,C 90.000,E1 290.120} C_DIS
LIN {X -0.100,Y -661.717,Z 924.411,A 0.000,B 0.000,C 90.000,E1 289.993} C_DIS
LIN {X 0.157,Y -661.930,Z 924.410,A 0.000,B 0.000,C 90.000,E1 289.812} C_DIS
LIN {X 0.050,Y -662.510,Z 924.409,A 0.000,B 0.000,C 90.000,E1 289.577} C_DIS
LIN {X 0.064,Y -664.399,Z 924.406,A 0.000,B 0.000,C 90.000,E1 289.087} C_DIS
LIN {X 0.028,Y -671.836,Z 924.398,A 0.000,B 0.000,C 90.000,E1 287.638} C_DIS
LIN {X 0.092,Y -674.152,Z 924.395,A 0.000,B 0.000,C 90.000,E1 287.149} C_DIS
LIN {X -0.032,Y -676.192,Z 924.393,A 0.000,B 0.000,C 90.000,E1 286.677} C_DIS
LIN {X -0.086,Y -677.160,Z 924.391,A 0.000,B 0.000,C 90.000,E1 286.441} C_DIS
LIN {X -0.042,Y -679.590,Z 924.387,A 0.000,B 0.000,C 90.000,E1 285.717} C_DIS
LIN {X -0.161,Y -681.442,Z 924.383,A 0.000,B 0.000,C 90.000,E1 285.009} C_DIS
LIN {X -0.260,Y -683.044,Z 924.379,A 0.000,B 0.000,C 90.000,E1 284.300} C_DIS
LIN {X 0.301,Y -684.817,Z 924.374,A 0.000,B 0.000,C 90.000,E1 283.300} C_DIS
LIN {X 0.237,Y -685.870,Z 924.370,A 0.000,B 0.000,C 90.000,E1 282.591} C_DIS
LIN {X 0.176,Y -686.693,Z 924.366,A 0.000,B 0.000,C 90.000,E1 281.883} C_DIS
LIN {X -0.018,Y -687.184,Z 924.362,A 0.000,B 0.000,C 90.000,E1 281.186} C_DIS
LIN {X -0.055,Y -687.202,Z 924.360,A 0.000,B 0.000,C 90.000,E1 280.715} C_DIS
LIN {X -0.220,Y -686.857,Z 924.357,A 0.000,B 0.000,C 90.000,E1 280.254} C_DIS
LIN {X -0.241,Y -686.549,Z 924.356,A 0.000,B 0.000,C 90.000,E1 280.018} C_DIS
LIN {X 0.272,Y -685.691,Z 924.353,A 0.000,B 0.000,C 90.000,E1 279.500} C_DIS
LIN {X 0.216,Y -684.288,Z 924.350,A 0.000,B 0.000,C 90.000,E1 279.029} C_DIS
LIN {X 0.042,Y -682.456,Z 924.348,A 0.000,B 0.000,C 90.000,E1 278.568} C_DIS
LIN {X -0.139,Y -680.271,Z 924.345,A 0.000,B 0.000,C 90.000,E1 278.106} C_DIS
LIN {X 0.283,Y -676.693,Z 924.341,A 0.000,B 0.000,C 90.000,E1 277.352} C_DIS
LIN {X -0.090,Y -672.846,Z 924.337,A 0.000,B 0.000,C 90.000,E1 276.663} C_DIS
LIN {X -0.330,Y -670.103,Z 924.334,A 0.000,B 0.000,C 90.000,E1 276.201} C_DIS
LIN {X 0.160,Y -667.870,Z 924.332,A 0.000,B 0.000,C 90.000,E1 275.796} C_DIS
LIN {X -0.203,Y -663.559,Z 924.329,A 0.000,B 0.000,C 90.000,E1 275.220} C_DIS
LIN {X 0.153,Y -659.807,Z 924.326,A 0.000,B 0.000,C 90.000,E1 274.702} C_DIS
LIN {X -0.224,Y -655.739,Z 924.324,A 0.000,B 0.000,C 90.000,E1 274.245} C_DIS
LIN {X -0.029,Y -650.115,Z 924.320,A 0.000,B 0.000,C 90.000,E1 273.612} C_DIS
LIN {X 0.323,Y -645.214,Z 924.317,A 0.000,B 0.000,C 90.000,E1 273.094} C_DIS
LIN {X 0.277,Y -638.749,Z 924.314,A 0.000,B 0.000,C 90.000,E1 272.522} C_DIS
LIN {X -0.165,Y -631.735,Z 924.311,A 0.000,B 0.000,C 90.000,E1 272.007} C_DIS
LIN {X -0.175,Y -624.304,Z 924.308,A 0.000,B 0.000,C 90.000,E1 271.489} C_DIS
LIN {X 0.111,Y -616.376,Z 924.306,A 0.000,B 0.000,C 90.000,E1 270.974} C_DIS
LIN {X -0.041,Y -610.216,Z 924.304,A 0.000,B 0.000,C 90.000,E1 270.630} C_DIS
LIN {X -0.032,Y -603.543,Z 924.302,A 0.000,B 0.000,C 90.000,E1 270.286} C_DIS
LIN {X 0.222,Y -596.704,Z 924.300,A 0.000,B 0.000,C 90.000,E1 269.943} C_DIS
LIN {X -0.256,Y -591.403,Z 924.299,A 0.000,B 0.000,C 90.000,E1 269.771} C_DIS
LIN {X -0.029,Y -583.996,Z 924.297,A 0.000,B 0.000,C 90.000,E1 269.484} C_DIS
LIN {X -0.014,Y -578.189,Z 924.296,A 0.000,B 0.000,C 90.000,E1 269.312} C_DIS
LIN {X -0.096,Y -570.325,Z 924.295,A 0.000,B 0.000,C 90.000,E1 269.141} C_DIS
LIN {X -0.006,Y -564.219,Z 924.295,A 0.000,B 0.000,C 90.000,E1 269.026} C_DIS
LIN {X -0.060,Y -557.934,Z 924.294,A 0.000,B 0.000,C 90.000,E1 268.969} C_DIS
LIN {X 0.087,Y -552.411,Z 924.294,A 0.000,B 0.000,C 90.000,E1 268.912} C_DIS
LIN {X -0.023,Y -550.127,Z 924.294,A 0.000,B 0.000,C 90.000,E1 268.854} C_DIS
LIN {X -0.054,Y -550.101,Z 924.294,A 0.000,B 0.000,C 90.000,E1 268.854} C_DIS
LIN {X -0.189,Y -548.758,Z 924.293,A 0.000,B 0.000,C 90.000,E1 268.682} C_DIS
LIN {X 0.160,Y -545.142,Z 924.290,A 0.000,B 0.000,C 90.000,E1 268.224} C_DIS
LIN {X -0.074,Y -544.237,Z 924.290,A 0.000,B 0.000,C 90.000,E1 268.165} C_DIS
LIN {X -0.116,Y -544.205,Z 924.290,A 0.000,B 0.000,C 90.000,E1 268.165} C_DIS
LIN {X -0.124,Y -543.304,Z 924.287,A 0.000,B 0.000,C 90.000,E1 267.707} C_DIS
LIN {X -0.252,Y -540.073,Z 924.267,A 0.000,B 0.000,C 90.000,E1 264.033} C_DIS
LIN {X -0.065,Y -539.081,Z 924.259,A 0.000,B 0.000,C 90.000,E1 262.591} C_DIS
LIN {X 0.181,Y -538.023,Z 924.251,A 0.000,B 0.000,C 90.000,E1 261.141} C_DIS
LIN {X -0.183,Y -537.003,Z 924.245,A 0.000,B 0.000,C 90.000,E1 260.038} C_DIS
LIN {X 0.001,Y -535.991,Z 924.240,A 0.000,B 0.000,C 90.000,E1 259.162} C_DIS
LIN {X -0.135,Y -533.366,Z 924.229,A 0.000,B 0.000,C 90.000,E1 257.173} C_DIS
LIN {X -0.054,Y -530.493,Z 924.216,A 0.000,B 0.000,C 90.000,E1 254.866} C_DIS
LIN {X -0.108,Y -528.388,Z 924.206,A 0.000,B 0.000,C 90.000,E1 253.142} C_DIS
LIN {X -0.239,Y -526.993,Z 924.200,A 0.000,B 0.000,C 90.000,E1 252.000} C_DIS
LIN {X 0.108,Y -524.346,Z 924.189,A 0.000,B 0.000,C 90.000,E1 249.934} C_DIS
LIN {X -0.076,Y -522.088,Z 924.179,A 0.000,B 0.000,C 90.000,E1 248.209} C_DIS
LIN {X -0.135,Y -520.478,Z 924.172,A 0.000,B 0.000,C 90.000,E1 247.050} C_DIS
LIN {X -0.168,Y -519.265,Z 924.168,A 0.000,B 0.000,C 90.000,E1 246.177} C_DIS
LIN {X -0.065,Y -516.496,Z 924.158,A 0.000,B 0.000,C 90.000,E1 244.409} C_DIS
LIN {X 0.076,Y -515.158,Z 924.153,A 0.000,B 0.000,C 90.000,E1 243.512} C_DIS
LIN {X 0.204,Y -512.772,Z 924.145,A 0.000,B 0.000,C 90.000,E1 242.025} C_DIS
LIN {X 0.193,Y -510.761,Z 924.138,A 0.000,B 0.000,C 90.000,E1 240.845} C_DIS
LIN {X 0.115,Y -507.555,Z 924.128,A 0.000,B 0.000,C 90.000,E1 239.076} C_DIS
LIN {X -0.151,Y -505.317,Z 924.122,A 0.000,B 0.000,C 90.000,E1 237.916} C_DIS
LIN {X 0.092,Y -503.463,Z 924.117,A 0.000,B 0.000,C 90.000,E1 236.993} C_DIS
LIN {X -0.138,Y -502.191,Z 924.113,A 0.000,B 0.000,C 90.000,E1 236.421} C_DIS
LIN {X 0.111,Y -496.750,Z 924.100,A 0.000,B 0.000,C 90.000,E1 233.989} C_DIS
LIN {X -0.168,Y -492.116,Z 924.088,A 0.000,B 0.000,C 90.000,E1 231.904} C_DIS
LIN {X 0.219,Y -489.392,Z 924.082,A 0.000,B 0.000,C 90.000,E1 230.642} C_DIS
LIN {X -0.152,Y -485.266,Z 924.071,A 0.000,B 0.000,C 90.000,E1 228.852} C_DIS
LIN {X 0.023,Y -481.140,Z 924.061,A 0.000,B 0.000,C 90.000,E1 226.986} C_DIS
LIN {X -0.130,Y -476.358,Z 924.049,A 0.000,B 0.000,C 90.000,E1 224.838} C_DIS
LIN {X 0.168,Y -472.217,Z 924.039,A 0.000,B 0.000,C 90.000,E1 222.933} C_DIS
LIN {X -0.032,Y -468.683,Z 924.030,A 0.000,B 0.000,C 90.000,E1 221.391} C_DIS
LIN {X 0.272,Y -463.220,Z 924.016,A 0.000,B 0.000,C 90.000,E1 218.830} C_DIS
LIN {X -0.076,Y -460.567,Z 924.009,A 0.000,B 0.000,C 90.000,E1 217.604} C_DIS
LIN {X 0.024,Y -456.449,Z 923.998,A 0.000,B 0.000,C 90.000,E1 215.678} C_DIS
LIN {X 0.040,Y -453.010,Z 923.989,A 0.000,B 0.000,C 90.000,E1 214.072} C_DIS
LIN {X -0.020,Y -449.303,Z 923.980,A 0.000,B 0.000,C 90.000,E1 212.467} C_DIS
LIN {X -0.094,Y -446.522,Z 923.973,A 0.000,B 0.000,C 90.000,E1 211.180} C_DIS
LIN {X 0.005,Y -442.923,Z 923.964,A 0.000,B 0.000,C 90.000,E1 209.539} C_DIS
LIN {X -0.006,Y -440.151,Z 923.957,A 0.000,B 0.000,C 90.000,E1 208.231} C_DIS
LIN {X 0.179,Y -435.800,Z 923.946,A 0.000,B 0.000,C 90.000,E1 206.232} C_DIS
LIN {X 0.086,Y -429.964,Z 923.931,A 0.000,B 0.000,C 90.000,E1 203.590} C_DIS
LIN {X 0.247,Y -426.309,Z 923.922,A 0.000,B 0.000,C 90.000,E1 201.897} C_DIS
LIN {X -0.172,Y -423.368,Z 923.914,A 0.000,B 0.000,C 90.000,E1 200.610} C_DIS
LIN {X 0.210,Y -417.250,Z 923.898,A 0.000,B 0.000,C 90.000,E1 197.511} C_DIS
LIN {X -0.207,Y -414.479,Z 923.890,A 0.000,B 0.000,C 90.000,E1 196.205} C_DIS
LIN {X -0.151,Y -411.738,Z 923.882,A 0.000,B 0.000,C 90.000,E1 194.828} C_DIS
LIN {X 0.164,Y -408.251,Z 923.873,A 0.000,B 0.000,C 90.000,E1 193.063} C_DIS
LIN {X -0.072,Y -404.775,Z 923.863,A 0.000,B 0.000,C 90.000,E1 191.366} C_DIS
LIN {X 0.012,Y -400.657,Z 923.852,A 0.000,B 0.000,C 90.000,E1 189.265} C_DIS
LIN {X -0.039,Y -397.879,Z 923.844,A 0.000,B 0.000,C 90.000,E1 187.871} C_DIS
LIN {X 0.201,Y -395.131,Z 923.836,A 0.000,B 0.000,C 90.000,E1 186.429} C_DIS
LIN {X -0.007,Y -389.248,Z 923.818,A 0.000,B 0.000,C 90.000,E1 183.269} C_DIS
LIN {X -0.148,Y -385.535,Z 923.806,A 0.000,B 0.000,C 90.000,E1 181.146} C_DIS
LIN {X 0.028,Y -380.866,Z 923.788,A 0.000,B 0.000,C 90.000,E1 177.879} C_DIS
LIN {X 0.062,Y -379.719,Z 923.782,A 0.000,B 0.000,C 90.000,E1 176.788} C_DIS
LIN {X -0.196,Y -379.409,Z 923.778,A 0.000,B 0.000,C 90.000,E1 176.102} C_DIS
LIN {X -0.089,Y -379.479,Z 923.773,A 0.000,B 0.000,C 90.000,E1 175.179} C_DIS
LIN {X 0.086,Y -380.151,Z 923.770,A 0.000,B 0.000,C 90.000,E1 174.609} C_DIS
LIN {X 0.055,Y -380.283,Z 923.769,A 0.000,B 0.000,C 90.000,E1 174.432} C_DIS
LIN {X -0.142,Y -381.063,Z 923.767,A 0.000,B 0.000,C 90.000,E1 174.090} C_DIS
LIN {X 0.144,Y -382.297,Z 923.765,A 0.000,B 0.000,C 90.000,E1 173.685} C_DIS
LIN {X 0.054,Y -383.693,Z 923.763,A 0.000,B 0.000,C 90.000,E1 173.337} C_DIS
LIN {X -0.076,Y -385.638,Z 923.761,A 0.000,B 0.000,C 90.000,E1 172.996} C_DIS
LIN {X -0.044,Y -387.597,Z 923.759,A 0.000,B 0.000,C 90.000,E1 172.704} C_DIS
LIN {X 0.189,Y -390.189,Z 923.758,A 0.000,B 0.000,C 90.000,E1 172.356} C_DIS
LIN {X -0.043,Y -394.715,Z 923.755,A 0.000,B 0.000,C 90.000,E1 171.951} C_DIS
LIN {X 0.071,Y -397.907,Z 923.754,A 0.000,B 0.000,C 90.000,E1 171.659} C_DIS
LIN {X -0.136,Y -411.032,Z 923.748,A 0.000,B 0.000,C 90.000,E1 170.735} C_DIS
LIN {X -0.019,Y -423.789,Z 923.743,A 0.000,B 0.000,C 90.000,E1 169.803} C_DIS
LIN {X 0.132,Y -433.265,Z 923.739,A 0.000,B 0.000,C 90.000,E1 169.050} C_DIS
LIN {X 0.099,Y -442.425,Z 923.735,A 0.000,B 0.000,C 90.000,E1 168.285} C_DIS
LIN {X -0.046,Y -449.930,Z 923.731,A 0.000,B 0.000,C 90.000,E1 167.645} C_DIS
LIN {X -0.201,Y -461.423,Z 923.725,A 0.000,B 0.000,C 90.000,E1 166.589} C_DIS
LIN {X 0.067,Y -466.860,Z 923.722,A 0.000,B 0.000,C 90.000,E1 165.992} C_DIS
LIN {X 0.006,Y -475.075,Z 923.717,A 0.000,B 0.000,C 90.000,E1 165.102} C_DIS
LIN {X 0.124,Y -485.490,Z 923.711,A 0.000,B 0.000,C 90.000,E1 163.866} C_DIS
LIN {X -0.237,Y -491.574,Z 923.706,A 0.000,B 0.000,C 90.000,E1 163.142} C_DIS
LIN {X -0.073,Y -497.370,Z 923.702,A 0.000,B 0.000,C 90.000,E1 162.362} C_DIS
LIN {X 0.222,Y -504.917,Z 923.696,A 0.000,B 0.000,C 90.000,E1 161.275} C_DIS
LIN {X 0.141,Y -512.228,Z 923.690,A 0.000,B 0.000,C 90.000,E1 160.242} C_DIS
LIN {X 0.061,Y -517.081,Z 923.686,A 0.000,B 0.000,C 90.000,E1 159.518} C_DIS
LIN {X 0.060,Y -520.074,Z 923.684,A 0.000,B 0.000,C 90.000,E1 159.082} C_DIS
LIN {X -0.154,Y -528.538,Z 923.677,A 0.000,B 0.000,C 90.000,E1 157.794} C_DIS
LIN {X 0.209,Y -532.163,Z 923.673,A 0.000,B 0.000,C 90.000,E1 157.177} C_DIS
LIN {X 0.118,Y -541.892,Z 923.665,A 0.000,B 0.000,C 90.000,E1 155.613} C_DIS
LIN {X 0.079,Y -548.670,Z 923.658,A 0.000,B 0.000,C 90.000,E1 154.485} C_DIS
LIN {X -0.122,Y -555.049,Z 923.652,A 0.000,B 0.000,C 90.000,E1 153.384} C_DIS
LIN {X 0.086,Y -558.771,Z 923.648,A 0.000,B 0.000,C 90.000,E1 152.666} C_DIS
LIN {X -0.134,Y -563.806,Z 923.643,A 0.000,B 0.000,C 90.000,E1 151.719} C_DIS
LIN {X 0.065,Y -569.960,Z 923.636,A 0.000,B 0.000,C 90.000,E1 150.461} C_DIS
LIN {X -0.085,Y -573.184,Z 923.632,A 0.000,B 0.000,C 90.000,E1 149.793} C_DIS
LIN {X 0.205,Y -576.842,Z 923.628,A 0.000,B 0.000,C 90.000,E1 148.948} C_DIS
LIN {X 0.348,Y -582.644,Z 923.620,A 0.000,B 0.000,C 90.000,E1 147.582} C_DIS
LIN {X -0.028,Y -589.364,Z 923.611,A 0.000,B 0.000,C 90.000,E1 146.008} C_DIS
LIN {X -0.372,Y -593.791,Z 923.605,A 0.000,B 0.000,C 90.000,E1 144.975} C_DIS
LIN {X -0.317,Y -597.764,Z 923.599,A 0.000,B 0.000,C 90.000,E1 143.909} C_DIS
LIN {X 0.041,Y -602.713,Z 923.592,A 0.000,B 0.000,C 90.000,E1 142.557} C_DIS
LIN {X 0.074,Y -609.686,Z 923.582,A 0.000,B 0.000,C 90.000,E1 140.723} C_DIS
LIN {X -0.319,Y -614.824,Z 923.575,A 0.000,B 0.000,C 90.000,E1 139.461} C_DIS
LIN {X -0.229,Y -619.892,Z 923.568,A 0.000,B 0.000,C 90.000,E1 138.162} C_DIS
LIN {X -0.225,Y -622.877,Z 923.563,A 0.000,B 0.000,C 90.000,E1 137.391} C_DIS
LIN {X -0.327,Y -627.165,Z 923.558,A 0.000,B 0.000,C 90.000,E1 136.377} C_DIS
LIN {X 0.064,Y -631.312,Z 923.552,A 0.000,B 0.000,C 90.000,E1 135.324} C_DIS
LIN {X 0.416,Y -636.403,Z 923.545,A 0.000,B 0.000,C 90.000,E1 134.028} C_DIS
LIN {X -0.059,Y -641.354,Z 923.538,A 0.000,B 0.000,C 90.000,E1 132.813} C_DIS
LIN {X -0.156,Y -649.182,Z 923.527,A 0.000,B 0.000,C 90.000,E1 130.825} C_DIS
LIN {X 0.162,Y -653.064,Z 923.521,A 0.000,B 0.000,C 90.000,E1 129.806} C_DIS
LIN {X -0.053,Y -660.612,Z 923.510,A 0.000,B 0.000,C 90.000,E1 127.855} C_DIS
LIN {X 0.048,Y -666.976,Z 923.501,A 0.000,B 0.000,C 90.000,E1 126.137} C_DIS
LIN {X -0.204,Y -671.291,Z 923.494,A 0.000,B 0.000,C 90.000,E1 124.945} C_DIS
LIN {X 0.168,Y -675.355,Z 923.487,A 0.000,B 0.000,C 90.000,E1 123.706} C_DIS
LIN {X -0.102,Y -677.553,Z 923.483,A 0.000,B 0.000,C 90.000,E1 123.007} C_DIS
LIN {X 0.005,Y -680.715,Z 923.477,A 0.000,B 0.000,C 90.000,E1 121.799} C_DIS
LIN {X -0.194,Y -681.875,Z 923.474,A 0.000,B 0.000,C 90.000,E1 121.337} C_DIS
LIN {X -0.219,Y -683.941,Z 923.469,A 0.000,B 0.000,C 90.000,E1 120.384} C_DIS
LIN {X -0.186,Y -685.326,Z 923.465,A 0.000,B 0.000,C 90.000,E1 119.667} C_DIS
LIN {X 0.084,Y -686.941,Z 923.459,A 0.000,B 0.000,C 90.000,E1 118.693} C_DIS
LIN {X -0.074,Y -687.673,Z 923.457,A 0.000,B 0.000,C 90.000,E1 118.231} C_DIS
LIN {X 0.228,Y -688.702,Z 923.452,A 0.000,B 0.000,C 90.000,E1 117.257} C_DIS
LIN {X -0.387,Y -689.195,Z 923.446,A 0.000,B 0.000,C 90.000,E1 116.360} C_DIS
LIN {X 0.312,Y -689.421,Z 923.442,A 0.000,B 0.000,C 90.000,E1 115.591} C_DIS
LIN {X 0.325,Y -689.439,Z 923.437,A 0.000,B 0.000,C 90.000,E1 114.643} C_DIS
LIN {X 0.106,Y -689.161,Z 923.433,A 0.000,B 0.000,C 90.000,E1 113.951} C_DIS
LIN {X -0.343,Y -688.755,Z 923.431,A 0.000,B 0.000,C 90.000,E1 113.515} C_DIS
LIN {X -0.160,Y -687.595,Z 923.428,A 0.000,B 0.000,C 90.000,E1 113.025} C_DIS
LIN {X 0.063,Y -686.776,Z 923.427,A 0.000,B 0.000,C 90.000,E1 112.770} C_DIS
LIN {X 0.127,Y -684.312,Z 923.425,A 0.000,B 0.000,C 90.000,E1 112.408} C_DIS
LIN {X 0.235,Y -683.612,Z 923.424,A 0.000,B 0.000,C 90.000,E1 112.280} C_DIS
LIN {X -0.295,Y -682.748,Z 923.423,A 0.000,B 0.000,C 90.000,E1 112.206} C_DIS
LIN {X -0.192,Y -681.456,Z 923.423,A 0.000,B 0.000,C 90.000,E1 112.078} C_DIS
LIN {X -0.035,Y -679.484,Z 923.422,A 0.000,B 0.000,C 90.000,E1 111.950} C_DIS
LIN {X 0.020,Y -674.855,Z 923.421,A 0.000,B 0.000,C 90.000,E1 111.770} C_DIS
LIN {X -0.095,Y -671.935,Z 923.420,A 0.000,B 0.000,C 90.000,E1 111.642} C_DIS
LIN {X 0.265,Y -669.806,Z 923.420,A 0.000,B 0.000,C 90.000,E1 111.535} C_DIS
LIN {X 0.180,Y -666.833,Z 923.419,A 0.000,B 0.000,C 90.000,E1 111.482} C_DIS
LIN {X 0.337,Y -662.089,Z 923.419,A 0.000,B 0.000,C 90.000,E1 111.408} C_DIS
LIN {X 0.082,Y -659.318,Z 923.419,A 0.000,B 0.000,C 90.000,E1 111.408} C_DIS
LIN {X -0.211,Y -642.632,Z 923.419,A 0.000,B 0.000,C 90.000,E1 111.408} C_DIS
LIN {X 0.146,Y -638.783,Z 923.419,A 0.000,B 0.000,C 90.000,E1 111.354} C_DIS
LIN {X -0.030,Y -628.710,Z 923.418,A 0.000,B 0.000,C 90.000,E1 111.227} C_DIS
LIN {X 0.232,Y -621.335,Z 923.417,A 0.000,B 0.000,C 90.000,E1 111.046} C_DIS
LIN {X -0.092,Y -614.120,Z 923.416,A 0.000,B 0.000,C 90.000,E1 110.865} C_DIS
LIN {X 0.307,Y -605.628,Z 923.414,A 0.000,B 0.000,C 90.000,E1 110.482} C_DIS
LIN {X -0.123,Y -598.820,Z 923.412,A 0.000,B 0.000,C 90.000,E1 110.174} C_DIS
LIN {X -0.221,Y -589.283,Z 923.409,A 0.000,B 0.000,C 90.000,E1 109.577} C_DIS
LIN {X 0.076,Y -578.949,Z 923.405,A 0.000,B 0.000,C 90.000,E1 108.852} C_DIS
LIN {X 0.003,Y -572.173,Z 923.403,A 0.000,B 0.000,C 90.000,E1 108.489} C_DIS
LIN {X 0.009,Y -566.655,Z 923.401,A 0.000,B 0.000,C 90.000,E1 108.236} C_DIS
LIN {X 0.096,Y -559.691,Z 923.400,A 0.000,B 0.000,C 90.000,E1 107.946} C_DIS
LIN {X 0.005,Y -556.480,Z 923.399,A 0.000,B 0.000,C 90.000,E1 107.819} C_DIS
LIN {X 0.004,Y -555.341,Z 923.399,A 0.000,B 0.000,C 90.000,E1 107.764} C_DIS
LIN {X 0.188,Y -554.002,Z 923.398,A 0.000,B 0.000,C 90.000,E1 107.638} C_DIS
LIN {X -0.015,Y -553.201,Z 923.398,A 0.000,B 0.000,C 90.000,E1 107.583} C_DIS
LIN {X -0.053,Y -553.183,Z 923.398,A 0.000,B 0.000,C 90.000,E1 107.583} C_DIS
LIN {X 0.006,Y -552.841,Z 923.397,A 0.000,B 0.000,C 90.000,E1 107.402} C_DIS
LIN {X 0.278,Y -552.802,Z 923.395,A 0.000,B 0.000,C 90.000,E1 107.094} C_DIS
LIN {X 0.193,Y -553.512,Z 923.386,A 0.000,B 0.000,C 90.000,E1 105.426} C_DIS
LIN {X -0.141,Y -554.133,Z 923.378,A 0.000,B 0.000,C 90.000,E1 104.064} C_DIS
LIN {X -0.216,Y -555.225,Z 923.367,A 0.000,B 0.000,C 90.000,E1 102.119} C_DIS
LIN {X 0.191,Y -556.871,Z 923.355,A 0.000,B 0.000,C 90.000,E1 99.849} C_DIS
LIN {X 0.234,Y -557.913,Z 923.347,A 0.000,B 0.000,C 90.000,E1 98.454} C_DIS
LIN {X 0.214,Y -558.928,Z 923.339,A 0.000,B 0.000,C 90.000,E1 97.068} C_DIS
LIN {X 0.001,Y -559.491,Z 923.335,A 0.000,B 0.000,C 90.000,E1 96.258} C_DIS
LIN {X 0.079,Y -560.494,Z 923.326,A 0.000,B 0.000,C 90.000,E1 94.588} C_DIS
LIN {X 0.128,Y -561.327,Z 923.316,A 0.000,B 0.000,C 90.000,E1 92.922} C_DIS
LIN {X 0.067,Y -561.978,Z 923.309,A 0.000,B 0.000,C 90.000,E1 91.547} C_DIS
LIN {X 0.005,Y -562.494,Z 923.301,A 0.000,B 0.000,C 90.000,E1 90.172} C_DIS
LIN {X -0.046,Y -562.840,Z 923.293,A 0.000,B 0.000,C 90.000,E1 88.797} C_DIS
LIN {X 0.151,Y -563.225,Z 923.283,A 0.000,B 0.000,C 90.000,E1 86.846} C_DIS
LIN {X 0.220,Y -563.492,Z 923.273,A 0.000,B 0.000,C 90.000,E1 85.184} C_DIS
LIN {X -0.033,Y -563.847,Z 923.263,A 0.000,B 0.000,C 90.000,E1 83.280} C_DIS
LIN {X 0.208,Y -564.153,Z 923.254,A 0.000,B 0.000,C 90.000,E1 81.602} C_DIS
LIN {X 0.057,Y -564.819,Z 923.243,A 0.000,B 0.000,C 90.000,E1 79.690} C_DIS
LIN {X 0.126,Y -565.747,Z 923.232,A 0.000,B 0.000,C 90.000,E1 77.757} C_DIS
LIN {X 0.213,Y -566.868,Z 923.221,A 0.000,B 0.000,C 90.000,E1 75.825} C_DIS
LIN {X 0.106,Y -567.668,Z 923.214,A 0.000,B 0.000,C 90.000,E1 74.464} C_DIS
LIN {X -0.328,Y -568.095,Z 923.209,A 0.000,B 0.000,C 90.000,E1 73.685} C_DIS
LIN {X -0.258,Y -568.760,Z 923.202,A 0.000,B 0.000,C 90.000,E1 72.308} C_DIS
LIN {X -0.037,Y -569.560,Z 923.191,A 0.000,B 0.000,C 90.000,E1 70.369} C_DIS
LIN {X 0.086,Y -569.877,Z 923.185,A 0.000,B 0.000,C 90.000,E1 69.263} C_DIS
LIN {X -0.174,Y -570.277,Z 923.177,A 0.000,B 0.000,C 90.000,E1 67.922} C_DIS
LIN {X 0.002,Y -570.496,Z 923.170,A 0.000,B 0.000,C 90.000,E1 66.538} C_DIS
LIN {X -0.215,Y -570.719,Z 923.161,A 0.000,B 0.000,C 90.000,E1 64.921} C_DIS
LIN {X 0.049,Y -570.881,Z 923.151,A 0.000,B 0.000,C 90.000,E1 63.256} C_DIS
LIN {X -0.188,Y -570.850,Z 923.142,A 0.000,B 0.000,C 90.000,E1 61.641} C_DIS
LIN {X 0.016,Y -570.841,Z 923.135,A 0.000,B 0.000,C 90.000,E1 60.255} C_DIS
LIN {X 0.103,Y -570.743,Z 923.129,A 0.000,B 0.000,C 90.000,E1 59.154} C_DIS
LIN {X 0.163,Y -570.653,Z 923.124,A 0.000,B 0.000,C 90.000,E1 58.329} C_DIS
LIN {X 0.173,Y -570.137,Z 923.117,A 0.000,B 0.000,C 90.000,E1 56.962} C_DIS
LIN {X 0.048,Y -569.644,Z 923.111,A 0.000,B 0.000,C 90.000,E1 55.881} C_DIS
LIN {X 0.104,Y -569.169,Z 923.106,A 0.000,B 0.000,C 90.000,E1 55.055} C_DIS
LIN {X -0.313,Y -568.598,Z 923.101,A 0.000,B 0.000,C 90.000,E1 54.276} C_DIS
LIN {X 0.061,Y -567.943,Z 923.097,A 0.000,B 0.000,C 90.000,E1 53.417} C_DIS
LIN {X -0.248,Y -566.767,Z 923.091,A 0.000,B 0.000,C 90.000,E1 52.351} C_DIS
LIN {X -0.226,Y -565.451,Z 923.085,A 0.000,B 0.000,C 90.000,E1 51.251} C_DIS
LIN {X 0.136,Y -563.772,Z 923.079,A 0.000,B 0.000,C 90.000,E1 50.114} C_DIS
LIN {X -0.087,Y -562.903,Z 923.076,A 0.000,B 0.000,C 90.000,E1 49.585} C_DIS
LIN {X -0.218,Y -561.357,Z 923.071,A 0.000,B 0.000,C 90.000,E1 48.771} C_DIS
LIN {X 0.001,Y -559.616,Z 923.066,A 0.000,B 0.000,C 90.000,E1 47.919} C_DIS
LIN {X 0.203,Y -557.645,Z 923.062,A 0.000,B 0.000,C 90.000,E1 47.067} C_DIS
LIN {X -0.022,Y -555.354,Z 923.057,A 0.000,B 0.000,C 90.000,E1 46.257} C_DIS
LIN {X -0.308,Y -553.742,Z 923.054,A 0.000,B 0.000,C 90.000,E1 45.729} C_DIS
LIN {X 0.209,Y -550.934,Z 923.049,A 0.000,B 0.000,C 90.000,E1 44.838} C_DIS
LIN {X 0.276,Y -548.952,Z 923.046,A 0.000,B 0.000,C 90.000,E1 44.271} C_DIS
LIN {X -0.041,Y -545.573,Z 923.042,A 0.000,B 0.000,C 90.000,E1 43.461} C_DIS
LIN {X 0.185,Y -543.853,Z 923.039,A 0.000,B 0.000,C 90.000,E1 43.014} C_DIS
LIN {X -0.006,Y -539.155,Z 923.034,A 0.000,B 0.000,C 90.000,E1 42.043} C_DIS
LIN {X 0.007,Y -536.239,Z 923.030,A 0.000,B 0.000,C 90.000,E1 41.472} C_DIS
LIN {X -0.225,Y -532.321,Z 923.026,A 0.000,B 0.000,C 90.000,E1 40.782} C_DIS
LIN {X -0.068,Y -529.798,Z 923.024,A 0.000,B 0.000,C 90.000,E1 40.334} C_DIS
LIN {X -0.057,Y -523.494,Z 923.018,A 0.000,B 0.000,C 90.000,E1 39.322} C_DIS
LIN {X -0.004,Y -518.701,Z 923.014,A 0.000,B 0.000,C 90.000,E1 38.588} C_DIS
LIN {X -0.121,Y -514.692,Z 923.011,A 0.000,B 0.000,C 90.000,E1 38.016} C_DIS
LIN {X -0.263,Y -510.502,Z 923.008,A 0.000,B 0.000,C 90.000,E1 37.443} C_DIS
LIN {X 0.170,Y -507.182,Z 923.005,A 0.000,B 0.000,C 90.000,E1 36.950} C_DIS
LIN {X -0.025,Y -502.508,Z 923.002,A 0.000,B 0.000,C 90.000,E1 36.377} C_DIS
LIN {X -0.045,Y -498.850,Z 923.000,A 0.000,B 0.000,C 90.000,E1 35.931} C_DIS
LIN {X 0.031,Y -494.948,Z 922.997,A 0.000,B 0.000,C 90.000,E1 35.471} C_DIS
LIN {X 0.069,Y -490.951,Z 922.995,A 0.000,B 0.000,C 90.000,E1 35.025} C_DIS
LIN {X -0.179,Y -483.941,Z 922.991,A 0.000,B 0.000,C 90.000,E1 34.326} C_DIS
LIN {X 0.130,Y -479.611,Z 922.988,A 0.000,B 0.000,C 90.000,E1 33.865} C_DIS
LIN {X -0.137,Y -470.893,Z 922.984,A 0.000,B 0.000,C 90.000,E1 33.086} C_DIS
LIN {X 0.025,Y -460.443,Z 922.979,A 0.000,B 0.000,C 90.000,E1 32.133} C_DIS
LIN {X -0.242,Y -448.210,Z 922.973,A 0.000,B 0.000,C 90.000,E1 31.131} C_DIS
LIN {X 0.105,Y -429.755,Z 922.964,A 0.000,B 0.000,C 90.000,E1 29.539} C_DIS
LIN {X 0.207,Y -411.558,Z 922.955,A 0.000,B 0.000,C 90.000,E1 27.897} C_DIS
LIN {X 0.198,Y -401.279,Z 922.950,A 0.000,B 0.000,C 90.000,E1 26.873} C_DIS
LIN {X 0.098,Y -396.837,Z 922.947,A 0.000,B 0.000,C 90.000,E1 26.411} C_DIS
LIN {X -0.041,Y -394.230,Z 922.945,A 0.000,B 0.000,C 90.000,E1 26.104} C_DIS
LIN {X 0.184,Y -391.296,Z 922.942,A 0.000,B 0.000,C 90.000,E1 25.591} C_DIS
LIN {X -0.068,Y -390.919,Z 922.942,A 0.000,B 0.000,C 90.000,E1 25.540} C_DIS
LIN {X -0.207,Y -389.365,Z 922.939,A 0.000,B 0.000,C 90.000,E1 25.027} C_DIS
LIN {X -0.031,Y -389.120,Z 922.938,A 0.000,B 0.000,C 90.000,E1 24.823} C_DIS
LIN {X 0.167,Y -388.617,Z 922.935,A 0.000,B 0.000,C 90.000,E1 24.259} C_DIS
LIN {X 0.128,Y -388.854,Z 922.929,A 0.000,B 0.000,C 90.000,E1 23.206} C_DIS
LIN {X -0.066,Y -392.844,Z 922.905,A 0.000,B 0.000,C 90.000,E1 18.960} C_DIS
LIN {X -0.171,Y -395.780,Z 922.892,A 0.000,B 0.000,C 90.000,E1 16.496} C_DIS
LIN {X 0.020,Y -399.875,Z 922.874,A 0.000,B 0.000,C 90.000,E1 13.300} C_DIS
LIN {X 0.106,Y -404.039,Z 922.858,A 0.000,B 0.000,C 90.000,E1 10.489} C_DIS
LIN {X 0.165,Y -408.048,Z 922.845,A 0.000,B 0.000,C 90.000,E1 8.049} C_DIS
LIN {X -0.169,Y -411.746,Z 922.833,A 0.000,B 0.000,C 90.000,E1 6.024} C_DIS
LIN {X -0.132,Y -415.081,Z 922.824,A 0.000,B 0.000,C 90.000,E1 4.302} C_DIS
LIN {X 0.106,Y -421.628,Z 922.807,A 0.000,B 0.000,C 90.000,E1 1.203} C_DIS
LIN {X -0.213,Y -425.738,Z 922.797,A 0.000,B 0.000,C 90.000,E1 359.484} C_DIS
LIN {X 0.032,Y -429.168,Z 922.790,A 0.000,B 0.000,C 90.000,E1 358.108} C_DIS
LIN {X 0.169,Y -431.311,Z 922.786,A 0.000,B 0.000,C 90.000,E1 357.421} C_DIS
LIN {X -0.190,Y -432.768,Z 922.784,A 0.000,B 0.000,C 90.000,E1 357.135} C_DIS
LIN {X 0.194,Y -433.969,Z 922.783,A 0.000,B 0.000,C 90.000,E1 356.849} C_DIS
LIN {X 0.090,Y -436.428,Z 922.781,A 0.000,B 0.000,C 90.000,E1 356.502} C_DIS
LIN {X -0.106,Y -437.127,Z 922.780,A 0.000,B 0.000,C 90.000,E1 356.445} C_DIS
LIN {X -0.200,Y -442.433,Z 922.778,A 0.000,B 0.000,C 90.000,E1 356.045} C_DIS
LIN {X 0.080,Y -448.282,Z 922.776,A 0.000,B 0.000,C 90.000,E1 355.698} C_DIS
LIN {X -0.064,Y -461.159,Z 922.773,A 0.000,B 0.000,C 90.000,E1 355.122} C_DIS
LIN {X 0.101,Y -471.209,Z 922.770,A 0.000,B 0.000,C 90.000,E1 354.609} C_DIS
LIN {X -0.080,Y -483.027,Z 922.767,A 0.000,B 0.000,C 90.000,E1 354.033} C_DIS
LIN {X 0.031,Y -494.691,Z 922.763,A 0.000,B 0.000,C 90.000,E1 353.394} C_DIS
LIN {X -0.107,Y -506.178,Z 922.760,A 0.000,B 0.000,C 90.000,E1 352.761} C_DIS
LIN {X -0.070,Y -515.604,Z 922.757,A 0.000,B 0.000,C 90.000,E1 352.186} C_DIS
LIN {X -0.014,Y -521.826,Z 922.754,A 0.000,B 0.000,C 90.000,E1 351.781} C_DIS
LIN {X -0.035,Y -530.892,Z 922.751,A 0.000,B 0.000,C 90.000,E1 351.141} C_DIS
LIN {X 0.055,Y -536.771,Z 922.748,A 0.000,B 0.000,C 90.000,E1 350.679} C_DIS
LIN {X -0.024,Y -543.756,Z 922.745,A 0.000,B 0.000,C 90.000,E1 350.095} C_DIS
LIN {X 0.104,Y -550.588,Z 922.742,A 0.000,B 0.000,C 90.000,E1 349.454} C_DIS
LIN {X -0.078,Y -556.993,Z 922.738,A 0.000,B 0.000,C 90.000,E1 348.814} C_DIS
LIN {X -0.149,Y -564.212,Z 922.733,A 0.000,B 0.000,C 90.000,E1 347.993} C_DIS
LIN {X 0.180,Y -568.731,Z 922.730,A 0.000,B 0.000,C 90.000,E1 347.409} C_DIS
LIN {X -0.013,Y -572.955,Z 922.727,A 0.000,B 0.000,C 90.000,E1 346.881} C_DIS
LIN {X 0.027,Y -578.934,Z 922.723,A 0.000,B 0.000,C 90.000,E1 346.061} C_DIS
LIN {X 0.270,Y -584.272,Z 922.718,A 0.000,B 0.000,C 90.000,E1 345.227} C_DIS
LIN {X 0.011,Y -589.361,Z 922.714,A 0.000,B 0.000,C 90.000,E1 344.448} C_DIS
LIN {X 0.073,Y -595.372,Z 922.708,A 0.000,B 0.000,C 90.000,E1 343.378} C_DIS
LIN {X 0.210,Y -600.976,Z 922.702,A 0.000,B 0.000,C 90.000,E1 342.308} C_DIS
LIN {X 0.030,Y -606.231,Z 922.696,A 0.000,B 0.000,C 90.000,E1 341.275} C_DIS
LIN {X -0.102,Y -611.912,Z 922.690,A 0.000,B 0.000,C 90.000,E1 340.115} C_DIS
LIN {X -0.119,Y -615.997,Z 922.685,A 0.000,B 0.000,C 90.000,E1 339.209} C_DIS
LIN {X -0.133,Y -621.589,Z 922.677,A 0.000,B 0.000,C 90.000,E1 337.922} C_DIS
LIN {X 0.178,Y -625.687,Z 922.672,A 0.000,B 0.000,C 90.000,E1 336.869} C_DIS
LIN {X -0.033,Y -629.420,Z 922.666,A 0.000,B 0.000,C 90.000,E1 335.869} C_DIS
LIN {X 0.142,Y -634.602,Z 922.658,A 0.000,B 0.000,C 90.000,E1 334.332} C_DIS
LIN {X -0.005,Y -637.135,Z 922.653,A 0.000,B 0.000,C 90.000,E1 333.589} C_DIS
LIN {X -0.364,Y -640.137,Z 922.648,A 0.000,B 0.000,C 90.000,E1 332.615} C_DIS
LIN {X -0.181,Y -642.342,Z 922.644,A 0.000,B 0.000,C 90.000,E1 331.847} C_DIS
LIN {X -0.160,Y -645.022,Z 922.638,A 0.000,B 0.000,C 90.000,E1 330.845} C_DIS
LIN {X -0.011,Y -648.106,Z 922.631,A 0.000,B 0.000,C 90.000,E1 329.587} C_DIS
LIN {X 0.187,Y -650.946,Z 922.624,A 0.000,B 0.000,C 90.000,E1 328.329} C_DIS
LIN {X -0.220,Y -652.983,Z 922.619,A 0.000,B 0.000,C 90.000,E1 327.375} C_DIS
LIN {X -0.058,Y -654.678,Z 922.613,A 0.000,B 0.000,C 90.000,E1 326.373} C_DIS
LIN {X -0.059,Y -656.165,Z 922.608,A 0.000,B 0.000,C 90.000,E1 325.388} C_DIS
LIN {X -0.035,Y -657.411,Z 922.602,A 0.000,B 0.000,C 90.000,E1 324.402} C_DIS
LIN {X 0.065,Y -658.309,Z 922.598,A 0.000,B 0.000,C 90.000,E1 323.657} C_DIS
LIN {X 0.055,Y -659.605,Z 922.591,A 0.000,B 0.000,C 90.000,E1 322.431} C_DIS
LIN {X -0.038,Y -660.660,Z 922.585,A 0.000,B 0.000,C 90.000,E1 321.215} C_DIS
LIN {X 0.021,Y -661.441,Z 922.579,A 0.000,B 0.000,C 90.000,E1 320.231} C_DIS
LIN {X -0.068,Y -662.838,Z 922.570,A 0.000,B 0.000,C 90.000,E1 318.528} C_DIS
LIN {X -0.098,Y -664.340,Z 922.561,A 0.000,B 0.000,C 90.000,E1 317.067} C_DIS
LIN {X 0.357,Y -665.241,Z 922.556,A 0.000,B 0.000,C 90.000,E1 316.053} C_DIS
LIN {X 0.341,Y -667.141,Z 922.543,A 0.000,B 0.000,C 90.000,E1 313.623} C_DIS
LIN {X 0.396,Y -669.062,Z 922.532,A 0.000,B 0.000,C 90.000,E1 311.676} C_DIS
LIN {X 0.045,Y -670.565,Z 922.522,A 0.000,B 0.000,C 90.000,E1 310.011} C_DIS
LIN {X 0.138,Y -671.391,Z 922.517,A 0.000,B 0.000,C 90.000,E1 309.036} C_DIS
LIN {X 0.346,Y -672.299,Z 922.510,A 0.000,B 0.000,C 90.000,E1 307.810} C_DIS
LIN {X 0.043,Y -672.976,Z 922.505,A 0.000,B 0.000,C 90.000,E1 306.870} C_DIS
LIN {X -0.119,Y -673.490,Z 922.498,A 0.000,B 0.000,C 90.000,E1 305.678} C_DIS
LIN {X 0.113,Y -674.012,Z 922.492,A 0.000,B 0.000,C 90.000,E1 304.452} C_DIS
LIN {X 0.147,Y -674.571,Z 922.485,A 0.000,B 0.000,C 90.000,E1 303.245} C_DIS
LIN {X 0.165,Y -675.367,Z 922.477,A 0.000,B 0.000,C 90.000,E1 301.799} C_DIS
LIN {X 0.124,Y -679.089,Z 922.454,A 0.000,B 0.000,C 90.000,E1 297.719} C_DIS
LIN {X 0.012,Y -682.503,Z 922.441,A 0.000,B 0.000,C 90.000,E1 295.335} C_DIS
LIN {X 0.149,Y -684.174,Z 922.434,A 0.000,B 0.000,C 90.000,E1 294.131} C_DIS
LIN {X -0.122,Y -684.911,Z 922.430,A 0.000,B 0.000,C 90.000,E1 293.439} C_DIS
LIN {X 0.030,Y -685.212,Z 922.428,A 0.000,B 0.000,C 90.000,E1 292.950} C_DIS
LIN {X 0.190,Y -685.210,Z 922.425,A 0.000,B 0.000,C 90.000,E1 292.461} C_DIS
LIN {X 0.400,Y -684.760,Z 922.424,A 0.000,B 0.000,C 90.000,E1 292.206} C_DIS
LIN {X -0.076,Y -683.326,Z 922.421,A 0.000,B 0.000,C 90.000,E1 291.770} C_DIS
LIN {X -0.227,Y -682.786,Z 922.420,A 0.000,B 0.000,C 90.000,E1 291.663} C_DIS
LIN {X -0.125,Y -681.953,Z 922.420,A 0.000,B 0.000,C 90.000,E1 291.535} C_DIS
LIN {X -0.025,Y -680.718,Z 922.419,A 0.000,B 0.000,C 90.000,E1 291.408} C_DIS
LIN {X -0.321,Y -676.706,Z 922.417,A 0.000,B 0.000,C 90.000,E1 291.099} C_DIS
LIN {X 0.064,Y -674.732,Z 922.416,A 0.000,B 0.000,C 90.000,E1 290.918} C_DIS
LIN {X 0.295,Y -662.745,Z 922.413,A 0.000,B 0.000,C 90.000,E1 290.248} C_DIS
LIN {X -0.055,Y -661.781,Z 922.412,A 0.000,B 0.000,C 90.000,E1 290.174} C_DIS
LIN {X -0.098,Y -661.760,Z 922.412,A 0.000,B 0.000,C 90.000,E1 290.174} C_DIS
LIN {X -0.078,Y -661.634,Z 922.411,A 0.000,B 0.000,C 90.000,E1 289.993} C_DIS
LIN {X -0.071,Y -662.797,Z 922.408,A 0.000,B 0.000,C 90.000,E1 289.504} C_DIS
LIN {X -0.031,Y -664.485,Z 922.406,A 0.000,B 0.000,C 90.000,E1 289.087} C_DIS
LIN {X -0.064,Y -671.924,Z 922.398,A 0.000,B 0.000,C 90.000,E1 287.638} C_DIS
LIN {X 0.000,Y -674.220,Z 922.395,A 0.000,B 0.000,C 90.000,E1 287.149} C_DIS
LIN {X -0.177,Y -677.191,Z 922.391,A 0.000,B 0.000,C 90.000,E1 286.441} C_DIS
LIN {X -0.134,Y -679.610,Z 922.387,A 0.000,B 0.000,C 90.000,E1 285.717} C_DIS
LIN {X -0.253,Y -681.460,Z 922.383,A 0.000,B 0.000,C 90.000,E1 285.009} C_DIS
LIN {X -0.351,Y -683.030,Z 922.379,A 0.000,B 0.000,C 90.000,E1 284.300} C_DIS
LIN {X 0.210,Y -684.829,Z 922.374,A 0.000,B 0.000,C 90.000,E1 283.300} C_DIS
LIN {X 0.124,Y -686.208,Z 922.369,A 0.000,B 0.000,C 90.000,E1 282.355} C_DIS
LIN {X -0.075,Y -686.860,Z 922.365,A 0.000,B 0.000,C 90.000,E1 281.658} C_DIS
LIN {X -0.110,Y -687.153,Z 922.362,A 0.000,B 0.000,C 90.000,E1 281.186} C_DIS
LIN {X -0.148,Y -687.203,Z 922.359,A 0.000,B 0.000,C 90.000,E1 280.715} C_DIS
LIN {X -0.312,Y -686.819,Z 922.357,A 0.000,B 0.000,C 90.000,E1 280.254} C_DIS
LIN {X 0.319,Y -686.096,Z 922.354,A 0.000,B 0.000,C 90.000,E1 279.726} C_DIS
LIN {X 0.180,Y -685.671,Z 922.353,A 0.000,B 0.000,C 90.000,E1 279.500} C_DIS
LIN {X 0.124,Y -684.267,Z 922.350,A 0.000,B 0.000,C 90.000,E1 279.029} C_DIS
LIN {X -0.050,Y -682.426,Z 922.348,A 0.000,B 0.000,C 90.000,E1 278.568} C_DIS
LIN {X -0.231,Y -680.267,Z 922.345,A 0.000,B 0.000,C 90.000,E1 278.106} C_DIS
LIN {X 0.176,Y -677.269,Z 922.342,A 0.000,B 0.000,C 90.000,E1 277.473} C_DIS
LIN {X -0.186,Y -672.802,Z 922.337,A 0.000,B 0.000,C 90.000,E1 276.663} C_DIS
LIN {X 0.241,Y -670.027,Z 922.334,A 0.000,B 0.000,C 90.000,E1 276.144} C_DIS
LIN {X 0.064,Y -667.778,Z 922.332,A 0.000,B 0.000,C 90.000,E1 275.796} C_DIS
LIN {X -0.298,Y -663.463,Z 922.329,A 0.000,B 0.000,C 90.000,E1 275.220} C_DIS
LIN {X 0.058,Y -659.710,Z 922.326,A 0.000,B 0.000,C 90.000,E1 274.702} C_DIS
LIN {X -0.320,Y -655.664,Z 922.323,A 0.000,B 0.000,C 90.000,E1 274.245} C_DIS
LIN {X -0.020,Y -651.236,Z 922.321,A 0.000,B 0.000,C 90.000,E1 273.726} C_DIS
LIN {X 0.250,Y -645.112,Z 922.317,A 0.000,B 0.000,C 90.000,E1 273.094} C_DIS
LIN {X 0.114,Y -638.510,Z 922.314,A 0.000,B 0.000,C 90.000,E1 272.522} C_DIS
LIN {X -0.250,Y -631.526,Z 922.311,A 0.000,B 0.000,C 90.000,E1 272.007} C_DIS
LIN {X -0.193,Y -624.142,Z 922.308,A 0.000,B 0.000,C 90.000,E1 271.489} C_DIS
LIN {X 0.119,Y -616.217,Z 922.306,A 0.000,B 0.000,C 90.000,E1 270.974} C_DIS
LIN {X 0.015,Y -610.046,Z 922.304,A 0.000,B 0.000,C 90.000,E1 270.630} C_DIS
LIN {X 0.039,Y -603.353,Z 922.302,A 0.000,B 0.000,C 90.000,E1 270.286} C_DIS
LIN {X -0.084,Y -598.289,Z 922.300,A 0.000,B 0.000,C 90.000,E1 270.057} C_DIS
LIN {X -0.170,Y -591.139,Z 922.299,A 0.000,B 0.000,C 90.000,E1 269.771} C_DIS
LIN {X 0.104,Y -583.737,Z 922.297,A 0.000,B 0.000,C 90.000,E1 269.484} C_DIS
LIN {X 0.147,Y -578.033,Z 922.296,A 0.000,B 0.000,C 90.000,E1 269.312} C_DIS
LIN {X 0.078,Y -570.047,Z 922.295,A 0.000,B 0.000,C 90.000,E1 269.141} C_DIS
LIN {X 0.173,Y -563.741,Z 922.295,A 0.000,B 0.000,C 90.000,E1 269.026} C_DIS
LIN {X 0.180,Y -558.068,Z 922.294,A 0.000,B 0.000,C 90.000,E1 268.969} C_DIS
LIN {X -0.227,Y -552.437,Z 922.294,A 0.000,B 0.000,C 90.000,E1 268.969} C_DIS
LIN {X -0.153,Y -548.827,Z 922.294,A 0.000,B 0.000,C 90.000,E1 268.854} C_DIS
LIN {X -0.184,Y -548.776,Z 922.294,A 0.000,B 0.000,C 90.000,E1 268.854} C_DIS
LIN {X -0.125,Y -547.535,Z 922.293,A 0.000,B 0.000,C 90.000,E1 268.682} C_DIS
LIN {X -0.128,Y -544.531,Z 922.291,A 0.000,B 0.000,C 90.000,E1 268.339} C_DIS
LIN {X -0.170,Y -544.509,Z 922.291,A 0.000,B 0.000,C 90.000,E1 268.339} C_DIS
LIN {X -0.228,Y -543.344,Z 922.287,A 0.000,B 0.000,C 90.000,E1 267.764} C_DIS
LIN {X 0.187,Y -540.100,Z 922.267,A 0.000,B 0.000,C 90.000,E1 264.033} C_DIS
LIN {X -0.158,Y -539.296,Z 922.261,A 0.000,B 0.000,C 90.000,E1 262.932} C_DIS
LIN {X 0.021,Y -538.240,Z 922.253,A 0.000,B 0.000,C 90.000,E1 261.489} C_DIS
LIN {X 0.190,Y -537.246,Z 922.246,A 0.000,B 0.000,C 90.000,E1 260.330} C_DIS
LIN {X -0.090,Y -536.017,Z 922.240,A 0.000,B 0.000,C 90.000,E1 259.218} C_DIS
LIN {X 0.143,Y -534.474,Z 922.234,A 0.000,B 0.000,C 90.000,E1 258.049} C_DIS
LIN {X -0.171,Y -533.085,Z 922.227,A 0.000,B 0.000,C 90.000,E1 256.937} C_DIS
LIN {X -0.270,Y -530.565,Z 922.216,A 0.000,B 0.000,C 90.000,E1 254.936} C_DIS
LIN {X -0.180,Y -528.446,Z 922.207,A 0.000,B 0.000,C 90.000,E1 253.196} C_DIS
LIN {X 0.195,Y -527.062,Z 922.200,A 0.000,B 0.000,C 90.000,E1 252.000} C_DIS
LIN {X -0.131,Y -524.443,Z 922.189,A 0.000,B 0.000,C 90.000,E1 250.007} C_DIS
LIN {X 0.164,Y -522.145,Z 922.179,A 0.000,B 0.000,C 90.000,E1 248.230} C_DIS
LIN {X -0.180,Y -520.549,Z 922.173,A 0.000,B 0.000,C 90.000,E1 247.102} C_DIS
LIN {X -0.065,Y -518.867,Z 922.166,A 0.000,B 0.000,C 90.000,E1 245.921} C_DIS
LIN {X -0.097,Y -516.579,Z 922.158,A 0.000,B 0.000,C 90.000,E1 244.460} C_DIS
LIN {X 0.048,Y -515.276,Z 922.153,A 0.000,B 0.000,C 90.000,E1 243.563} C_DIS
LIN {X 0.289,Y -512.394,Z 922.143,A 0.000,B 0.000,C 90.000,E1 241.769} C_DIS
LIN {X 0.270,Y -510.317,Z 922.137,A 0.000,B 0.000,C 90.000,E1 240.589} C_DIS
LIN {X 0.110,Y -507.647,Z 922.129,A 0.000,B 0.000,C 90.000,E1 239.125} C_DIS
LIN {X 0.011,Y -505.412,Z 922.122,A 0.000,B 0.000,C 90.000,E1 237.946} C_DIS
LIN {X 0.101,Y -503.607,Z 922.117,A 0.000,B 0.000,C 90.000,E1 237.041} C_DIS
LIN {X -0.102,Y -501.624,Z 922.112,A 0.000,B 0.000,C 90.000,E1 236.167} C_DIS
LIN {X -0.022,Y -497.597,Z 922.102,A 0.000,B 0.000,C 90.000,E1 234.356} C_DIS
LIN {X -0.140,Y -493.555,Z 922.092,A 0.000,B 0.000,C 90.000,E1 232.557} C_DIS
LIN {X 0.117,Y -490.287,Z 922.083,A 0.000,B 0.000,C 90.000,E1 231.009} C_DIS
LIN {X 0.278,Y -485.427,Z 922.072,A 0.000,B 0.000,C 90.000,E1 228.852} C_DIS
LIN {X -0.095,Y -480.667,Z 922.060,A 0.000,B 0.000,C 90.000,E1 226.743} C_DIS
LIN {X 0.188,Y -477.288,Z 922.051,A 0.000,B 0.000,C 90.000,E1 225.162} C_DIS
LIN {X 0.027,Y -471.735,Z 922.037,A 0.000,B 0.000,C 90.000,E1 222.690} C_DIS
LIN {X -0.113,Y -464.722,Z 922.020,A 0.000,B 0.000,C 90.000,E1 219.564} C_DIS
LIN {X -0.008,Y -460.733,Z 922.009,A 0.000,B 0.000,C 90.000,E1 217.649} C_DIS
LIN {X 0.085,Y -456.612,Z 921.999,A 0.000,B 0.000,C 90.000,E1 215.724} C_DIS
LIN {X 0.097,Y -453.217,Z 921.990,A 0.000,B 0.000,C 90.000,E1 214.119} C_DIS
LIN {X 0.085,Y -450.241,Z 921.982,A 0.000,B 0.000,C 90.000,E1 212.832} C_DIS
LIN {X 0.108,Y -446.722,Z 921.974,A 0.000,B 0.000,C 90.000,E1 211.209} C_DIS
LIN {X 0.053,Y -443.097,Z 921.964,A 0.000,B 0.000,C 90.000,E1 209.589} C_DIS
LIN {X -0.125,Y -439.592,Z 921.955,A 0.000,B 0.000,C 90.000,E1 207.975} C_DIS
LIN {X 0.048,Y -435.252,Z 921.944,A 0.000,B 0.000,C 90.000,E1 205.976} C_DIS
LIN {X -0.063,Y -429.415,Z 921.930,A 0.000,B 0.000,C 90.000,E1 203.334} C_DIS
LIN {X -0.119,Y -425.087,Z 921.918,A 0.000,B 0.000,C 90.000,E1 201.334} C_DIS
LIN {X 0.119,Y -417.444,Z 921.898,A 0.000,B 0.000,C 90.000,E1 197.583} C_DIS
LIN {X -0.025,Y -414.015,Z 921.888,A 0.000,B 0.000,C 90.000,E1 195.898} C_DIS
LIN {X -0.089,Y -411.232,Z 921.881,A 0.000,B 0.000,C 90.000,E1 194.537} C_DIS
LIN {X -0.178,Y -407.781,Z 921.871,A 0.000,B 0.000,C 90.000,E1 192.827} C_DIS
LIN {X -0.025,Y -404.250,Z 921.862,A 0.000,B 0.000,C 90.000,E1 191.074} C_DIS
LIN {X 0.053,Y -400.871,Z 921.852,A 0.000,B 0.000,C 90.000,E1 189.321} C_DIS
LIN {X -0.092,Y -396.735,Z 921.840,A 0.000,B 0.000,C 90.000,E1 187.239} C_DIS
LIN {X -0.176,Y -390.661,Z 921.823,A 0.000,B 0.000,C 90.000,E1 184.069} C_DIS
LIN {X -0.118,Y -388.221,Z 921.815,A 0.000,B 0.000,C 90.000,E1 182.636} C_DIS
LIN {X 0.151,Y -382.885,Z 921.797,A 0.000,B 0.000,C 90.000,E1 179.370} C_DIS
LIN {X 0.098,Y -379.628,Z 921.783,A 0.000,B 0.000,C 90.000,E1 176.849} C_DIS
LIN {X -0.137,Y -379.198,Z 921.779,A 0.000,B 0.000,C 90.000,E1 176.159} C_DIS
LIN {X -0.066,Y -378.986,Z 921.774,A 0.000,B 0.000,C 90.000,E1 175.241} C_DIS
LIN {X 0.100,Y -379.362,Z 921.771,A 0.000,B 0.000,C 90.000,E1 174.837} C_DIS
LIN {X -0.070,Y -379.692,Z 921.768,A 0.000,B 0.000,C 90.000,E1 174.318} C_DIS
LIN {X -0.139,Y -379.930,Z 921.767,A 0.000,B 0.000,C 90.000,E1 174.147} C_DIS
LIN {X 0.183,Y -380.958,Z 921.765,A 0.000,B 0.000,C 90.000,E1 173.628} C_DIS
LIN {X -0.081,Y -383.289,Z 921.761,A 0.000,B 0.000,C 90.000,E1 173.053} C_DIS
LIN {X 0.099,Y -385.589,Z 921.759,A 0.000,B 0.000,C 90.000,E1 172.591} C_DIS
LIN {X 0.086,Y -386.856,Z 921.758,A 0.000,B 0.000,C 90.000,E1 172.413} C_DIS
LIN {X 0.125,Y -391.358,Z 921.755,A 0.000,B 0.000,C 90.000,E1 171.894} C_DIS
LIN {X 0.080,Y -397.164,Z 921.752,A 0.000,B 0.000,C 90.000,E1 171.376} C_DIS
LIN {X 0.103,Y -415.825,Z 921.745,A 0.000,B 0.000,C 90.000,E1 170.038} C_DIS
LIN {X -0.206,Y -420.551,Z 921.743,A 0.000,B 0.000,C 90.000,E1 169.746} C_DIS
LIN {X 0.084,Y -431.673,Z 921.738,A 0.000,B 0.000,C 90.000,E1 168.870} C_DIS
LIN {X 0.114,Y -439.367,Z 921.735,A 0.000,B 0.000,C 90.000,E1 168.229} C_DIS
LIN {X 0.061,Y -446.952,Z 921.731,A 0.000,B 0.000,C 90.000,E1 167.589} C_DIS
LIN {X -0.063,Y -452.803,Z 921.728,A 0.000,B 0.000,C 90.000,E1 167.061} C_DIS
LIN {X -0.227,Y -463.148,Z 921.723,A 0.000,B 0.000,C 90.000,E1 166.117} C_DIS
LIN {X -0.111,Y -474.020,Z 921.716,A 0.000,B 0.000,C 90.000,E1 164.936} C_DIS
LIN {X 0.210,Y -484.396,Z 921.710,A 0.000,B 0.000,C 90.000,E1 163.685} C_DIS
LIN {X -0.117,Y -490.549,Z 921.705,A 0.000,B 0.000,C 90.000,E1 162.960} C_DIS
LIN {X -0.214,Y -495.205,Z 921.702,A 0.000,B 0.000,C 90.000,E1 162.362} C_DIS
LIN {X 0.048,Y -502.991,Z 921.696,A 0.000,B 0.000,C 90.000,E1 161.275} C_DIS
LIN {X 0.230,Y -511.295,Z 921.689,A 0.000,B 0.000,C 90.000,E1 160.061} C_DIS
LIN {X 0.068,Y -519.270,Z 921.683,A 0.000,B 0.000,C 90.000,E1 158.901} C_DIS
LIN {X -0.321,Y -528.744,Z 921.675,A 0.000,B 0.000,C 90.000,E1 157.486} C_DIS
LIN {X -0.243,Y -540.292,Z 921.664,A 0.000,B 0.000,C 90.000,E1 155.613} C_DIS
LIN {X -0.074,Y -547.165,Z 921.658,A 0.000,B 0.000,C 90.000,E1 154.460} C_DIS
LIN {X -0.042,Y -553.638,Z 921.652,A 0.000,B 0.000,C 90.000,E1 153.332} C_DIS
LIN {X 0.148,Y -557.404,Z 921.648,A 0.000,B 0.000,C 90.000,E1 152.615} C_DIS
LIN {X 0.077,Y -563.175,Z 921.642,A 0.000,B 0.000,C 90.000,E1 151.513} C_DIS
LIN {X 0.081,Y -568.684,Z 921.636,A 0.000,B 0.000,C 90.000,E1 150.411} C_DIS
LIN {X 0.034,Y -573.218,Z 921.630,A 0.000,B 0.000,C 90.000,E1 149.459} C_DIS
LIN {X -0.183,Y -579.252,Z 921.623,A 0.000,B 0.000,C 90.000,E1 148.122} C_DIS
LIN {X -0.093,Y -583.292,Z 921.618,A 0.000,B 0.000,C 90.000,E1 147.168} C_DIS
LIN {X 0.164,Y -588.921,Z 921.610,A 0.000,B 0.000,C 90.000,E1 145.801} C_DIS
LIN {X -0.186,Y -593.336,Z 921.604,A 0.000,B 0.000,C 90.000,E1 144.769} C_DIS
LIN {X 0.094,Y -598.372,Z 921.597,A 0.000,B 0.000,C 90.000,E1 143.417} C_DIS
LIN {X -0.032,Y -601.397,Z 921.592,A 0.000,B 0.000,C 90.000,E1 142.637} C_DIS
LIN {X 0.315,Y -611.517,Z 921.578,A 0.000,B 0.000,C 90.000,E1 139.989} C_DIS
LIN {X -0.221,Y -617.684,Z 921.569,A 0.000,B 0.000,C 90.000,E1 138.485} C_DIS
LIN {X -0.085,Y -619.737,Z 921.566,A 0.000,B 0.000,C 90.000,E1 137.957} C_DIS
LIN {X -0.395,Y -621.737,Z 921.564,A 0.000,B 0.000,C 90.000,E1 137.472} C_DIS
LIN {X 0.107,Y -628.114,Z 921.555,A 0.000,B 0.000,C 90.000,E1 135.891} C_DIS
LIN {X 0.068,Y -632.224,Z 921.549,A 0.000,B 0.000,C 90.000,E1 134.879} C_DIS
LIN {X 0.086,Y -636.297,Z 921.544,A 0.000,B 0.000,C 90.000,E1 133.866} C_DIS
LIN {X 0.166,Y -640.324,Z 921.538,A 0.000,B 0.000,C 90.000,E1 132.852} C_DIS
LIN {X 0.146,Y -646.223,Z 921.530,A 0.000,B 0.000,C 90.000,E1 131.353} C_DIS
LIN {X 0.357,Y -651.136,Z 921.523,A 0.000,B 0.000,C 90.000,E1 130.092} C_DIS
LIN {X -0.263,Y -655.833,Z 921.516,A 0.000,B 0.000,C 90.000,E1 128.910} C_DIS
LIN {X 0.110,Y -660.589,Z 921.509,A 0.000,B 0.000,C 90.000,E1 127.649} C_DIS
LIN {X -0.282,Y -666.066,Z 921.501,A 0.000,B 0.000,C 90.000,E1 126.217} C_DIS
LIN {X 0.000,Y -670.382,Z 921.494,A 0.000,B 0.000,C 90.000,E1 124.978} C_DIS
LIN {X 0.217,Y -673.674,Z 921.489,A 0.000,B 0.000,C 90.000,E1 123.992} C_DIS
LIN {X 0.099,Y -676.638,Z 921.484,A 0.000,B 0.000,C 90.000,E1 123.038} C_DIS
LIN {X 0.021,Y -679.282,Z 921.478,A 0.000,B 0.000,C 90.000,E1 122.084} C_DIS
LIN {X -0.221,Y -681.054,Z 921.474,A 0.000,B 0.000,C 90.000,E1 121.386} C_DIS
LIN {X -0.019,Y -683.152,Z 921.469,A 0.000,B 0.000,C 90.000,E1 120.413} C_DIS
LIN {X 0.353,Y -684.555,Z 921.465,A 0.000,B 0.000,C 90.000,E1 119.667} C_DIS
LIN {X 0.012,Y -686.158,Z 921.460,A 0.000,B 0.000,C 90.000,E1 118.743} C_DIS
LIN {X 0.068,Y -687.204,Z 921.456,A 0.000,B 0.000,C 90.000,E1 118.025} C_DIS
LIN {X 0.046,Y -688.140,Z 921.451,A 0.000,B 0.000,C 90.000,E1 117.078} C_DIS
LIN {X 0.352,Y -688.578,Z 921.445,A 0.000,B 0.000,C 90.000,E1 116.104} C_DIS
LIN {X 0.125,Y -688.750,Z 921.441,A 0.000,B 0.000,C 90.000,E1 115.412} C_DIS
LIN {X 0.134,Y -688.701,Z 921.436,A 0.000,B 0.000,C 90.000,E1 114.463} C_DIS
LIN {X -0.037,Y -688.506,Z 921.433,A 0.000,B 0.000,C 90.000,E1 114.003} C_DIS
LIN {X 0.139,Y -688.121,Z 921.431,A 0.000,B 0.000,C 90.000,E1 113.515} C_DIS
LIN {X -0.317,Y -687.104,Z 921.428,A 0.000,B 0.000,C 90.000,E1 113.078} C_DIS
LIN {X -0.095,Y -686.335,Z 921.427,A 0.000,B 0.000,C 90.000,E1 112.823} C_DIS
LIN {X 0.086,Y -683.677,Z 921.424,A 0.000,B 0.000,C 90.000,E1 112.386} C_DIS
LIN {X -0.069,Y -682.961,Z 921.424,A 0.000,B 0.000,C 90.000,E1 112.280} C_DIS
LIN {X 0.035,Y -681.975,Z 921.423,A 0.000,B 0.000,C 90.000,E1 112.153} C_DIS
LIN {X 0.135,Y -680.487,Z 921.422,A 0.000,B 0.000,C 90.000,E1 112.025} C_DIS
LIN {X 0.299,Y -671.436,Z 921.420,A 0.000,B 0.000,C 90.000,E1 111.589} C_DIS
LIN {X 0.062,Y -669.293,Z 921.420,A 0.000,B 0.000,C 90.000,E1 111.535} C_DIS
LIN {X -0.366,Y -667.572,Z 921.419,A 0.000,B 0.000,C 90.000,E1 111.535} C_DIS
LIN {X -0.026,Y -659.808,Z 921.419,A 0.000,B 0.000,C 90.000,E1 111.408} C_DIS
LIN {X 0.236,Y -648.951,Z 921.419,A 0.000,B 0.000,C 90.000,E1 111.354} C_DIS
LIN {X 0.048,Y -640.943,Z 921.419,A 0.000,B 0.000,C 90.000,E1 111.354} C_DIS
LIN {X -0.007,Y -634.095,Z 921.418,A 0.000,B 0.000,C 90.000,E1 111.280} C_DIS
LIN {X 0.071,Y -627.860,Z 921.418,A 0.000,B 0.000,C 90.000,E1 111.173} C_DIS
LIN {X 0.140,Y -622.329,Z 921.417,A 0.000,B 0.000,C 90.000,E1 111.046} C_DIS
LIN {X 0.049,Y -614.984,Z 921.416,A 0.000,B 0.000,C 90.000,E1 110.844} C_DIS
LIN {X -0.220,Y -611.397,Z 921.415,A 0.000,B 0.000,C 90.000,E1 110.737} C_DIS
LIN {X 0.195,Y -604.880,Z 921.414,A 0.000,B 0.000,C 90.000,E1 110.429} C_DIS
LIN {X -0.247,Y -598.133,Z 921.412,A 0.000,B 0.000,C 90.000,E1 110.120} C_DIS
LIN {X 0.160,Y -586.512,Z 921.407,A 0.000,B 0.000,C 90.000,E1 109.322} C_DIS
